(* IEC 61131-3 sources: Summary-ETFA22/benchmark/PLCopen_safety, 34 files *)

(* ---- SFAntivalent.st ---- *)
PROGRAM Main
VAR_INPUT
    Activate : BOOL;
    SChannelNC : SAFEBOOL;
    SChannelNO : SAFEBOOL;
    DiscrepancyTime : TIME;
END_VAR
VAR
    SFAntivalent : SFAntivalent;
END_VAR
SFAntivalent(Activate:=Activate,SChannelNC:=SChannelNC,SChannelNO:=SChannelNO,DiscrepancyTime:=DiscrepancyTime);
END_PROGRAM

FUNCTION_BLOCK SFAntivalent
VAR_INPUT
    Activate : BOOL;
    SChannelNC : SAFEBOOL;
    SChannelNO : SAFEBOOL;
    DiscrepancyTime : TIME;
END_VAR
VAR
    IN : BOOL;
    PT : TIME;
    running : BOOL;
    Q : BOOL;
END_VAR
VAR_OUTPUT
    Ready : BOOL;
    SAntivalentOut : BOOL;
    Error : BOOL;
    DiagCode : WORD;
END_VAR

IF NOT Activate THEN
    DiagCode := 16#0000;
ELSE
    CASE DiagCode OF
    16#0000:
        IF Activate THEN
            DiagCode := 16#8001;
        END_IF;
    16#8001:
        IF SChannelNC AND SChannelNO THEN
            DiagCode := 16#8004;
            IN:=TRUE;
            PT:=DiscrepancyTime;
            IF NOT running AND NOT Q THEN
                running := TRUE;
            ELSIF running AND NOT Q THEN
                Q := NONDETERMINISTIC_BOOL();
                running := NOT Q;
            END_IF;
        ELSIF NOT SChannelNC AND NOT SChannelNO THEN
            DiagCode := 16#8014;
            IN:=TRUE;
            PT:=DiscrepancyTime;
            IF NOT running AND NOT Q THEN
                running := TRUE;
            ELSIF running AND NOT Q THEN
                Q := NONDETERMINISTIC_BOOL();
                running := NOT Q;
            END_IF;
        ELSIF SChannelNC AND NOT SChannelNO THEN
            DiagCode := 16#8000;
        END_IF;
    16#8004:
        IF Q THEN
            DiagCode := 16#C001;
        ELSIF NOT SChannelNC THEN
            DiagCode := 16#8001;
        ELSIF NOT SChannelNO THEN
            DiagCode := 16#8000;
        END_IF;
    16#C001,
    16#C002:
        IF NOT SChannelNC AND SChannelNO THEN
            DiagCode := 16#8001;
        END_IF;
    16#8014:
        IF Q THEN
            DiagCode := 16#C002;
        ELSIF SChannelNO THEN
            DiagCode := 16#8001;
        ELSIF SChannelNC THEN
            DiagCode := 16#8000;
        END_IF;
    16#C003:
        IF NOT SChannelNC AND SChannelNO THEN
            DiagCode := 16#8001;
        END_IF;
    16#8005:
        IF Q THEN
            DiagCode := 16#C003;
        ELSIF NOT SChannelNC AND SChannelNO THEN
            DiagCode := 16#8001;
        END_IF;
    16#8000:
        IF NOT SChannelNC OR SChannelNO THEN
            DiagCode := 16#8005;
            IN:=TRUE;
            PT:=DiscrepancyTime;
            IF NOT running AND NOT Q THEN
                running := TRUE;
            ELSIF running AND NOT Q THEN
                Q := NONDETERMINISTIC_BOOL();
                running := NOT Q;
            END_IF;
        ELSIF NOT SChannelNC AND SChannelNO THEN
            DiagCode := 16#8001;
        END_IF;
    END_CASE;
END_IF;

CASE DiagCode OF
16#0000:
    Q := FALSE;
    running := FALSE;
    Ready := FALSE;
    Error := FALSE;
    SAntivalentOut:= FALSE;
16#8000:
    Q := FALSE;
    running := FALSE;
    Ready := TRUE;
    Error := FALSE;
    SAntivalentOut := TRUE;
16#8001:
    IN:=FALSE;
    PT:=DiscrepancyTime;
    Q := FALSE;
    running := FALSE;
    Ready := TRUE;
    Error := FALSE;
    SAntivalentOut:= FALSE;
16#8004,
16#8014,
16#8005:
    IN := TRUE;
    PT := DiscrepancyTime;
    IF NOT running AND NOT Q THEN
        running := TRUE;
    ELSIF running AND NOT Q THEN
        Q := NONDETERMINISTIC_BOOL();
        running := NOT Q;
    END_IF;
    Ready := TRUE;
    Error := FALSE;
    SAntivalentOut:= FALSE;
16#C001,
16#C002,
16#C003:
    IN := FALSE;
    PT := DiscrepancyTime;
    Q := FALSE;
    running := FALSE;
    Ready := TRUE;
    Error := TRUE;
    SAntivalentOut:= FALSE;
END_CASE;
END_FUNCTION_BLOCK

(* ---- SFAntivalent_CAP.st ---- *)
PROGRAM Main
VAR_INPUT
    Activate : BOOL;
    SChannelNC : SAFEBOOL;
    SChannelNO : SAFEBOOL;
    DiscrepancyTime : TIME;
END_VAR
VAR
    SFAntivalent : SFAntivalent;
END_VAR
SFAntivalent(Activate:=Activate,SChannelNC:=SChannelNC,SChannelNO:=SChannelNO,DiscrepancyTime:=DiscrepancyTime);
END_PROGRAM

FUNCTION_BLOCK SFAntivalent
VAR_INPUT
    Activate : BOOL;
    SChannelNC : SAFEBOOL;
    SChannelNO : SAFEBOOL;
    DiscrepancyTime : TIME;
END_VAR
VAR
    IN : BOOL;
    PT : TIME;
    running : BOOL;
    Q : BOOL;
END_VAR
VAR_OUTPUT
    Ready : BOOL;
    SAntivalentOut : BOOL;
    Error : BOOL;
    DiagCode : WORD;
END_VAR

IF NOT Activate THEN
    DiagCode := 16#0000;
ELSE
    CASE DiagCode OF
    change(16#0000, 16#0000):
        IF Activate THEN
            DiagCode := change(16#8001, 16#8001);
        END_IF;
    16#8001:
        IF SChannelNC AND SChannelNO THEN
            DiagCode := 16#8004;
            IN:=TRUE;
            PT:=DiscrepancyTime;
            IF NOT running AND NOT Q THEN
                running := TRUE;
            ELSIF running AND NOT Q THEN
                Q := NONDETERMINISTIC_BOOL();
                running := NOT Q;
            END_IF;
        ELSIF NOT SChannelNC AND NOT SChannelNO THEN
            DiagCode := 16#8014;
            IN:=TRUE;
            PT:=DiscrepancyTime;
            IF NOT running AND NOT Q THEN
                running := TRUE;
            ELSIF running AND NOT Q THEN
                Q := NONDETERMINISTIC_BOOL();
                running := NOT Q;
            END_IF;
        ELSIF SChannelNC AND NOT SChannelNO THEN
            DiagCode := 16#8000;
        END_IF;
    16#8004:
        IF Q THEN
            DiagCode := 16#C001;
        ELSIF NOT SChannelNC THEN
            DiagCode := 16#8001;
        ELSIF NOT SChannelNO THEN
            DiagCode := 16#8000;
        END_IF;
    16#C001,
    16#C002:
        IF NOT SChannelNC AND SChannelNO THEN
            DiagCode := 16#8001;
        END_IF;
    16#8014:
        IF Q THEN
            DiagCode := 16#C002;
        ELSIF SChannelNO THEN
            DiagCode := 16#8001;
        ELSIF SChannelNC THEN
            DiagCode := 16#8000;
        END_IF;
    16#C003:
        IF NOT SChannelNC AND SChannelNO THEN
            DiagCode := 16#8001;
        END_IF;
    16#8005:
        IF Q THEN
            DiagCode := 16#C003;
        ELSIF NOT SChannelNC AND SChannelNO THEN
            DiagCode := 16#8001;
        END_IF;
    16#8000:
        IF NOT SChannelNC OR SChannelNO THEN
            DiagCode := 16#8005;
            IN:=TRUE;
            PT:=DiscrepancyTime;
            IF NOT running AND NOT Q THEN
                running := TRUE;
            ELSIF running AND NOT Q THEN
                Q := NONDETERMINISTIC_BOOL();
                running := NOT Q;
            END_IF;
        ELSIF NOT SChannelNC AND SChannelNO THEN
            DiagCode := 16#8001;
        END_IF;
    END_CASE;
END_IF;

CASE DiagCode OF
16#0000:
    Q := FALSE;
    running := FALSE;
    Ready := FALSE;
    Error := FALSE;
    SAntivalentOut:= FALSE;
16#8000:
    Q := FALSE;
    running := FALSE;
    Ready := TRUE;
    Error := FALSE;
    SAntivalentOut := TRUE;
16#8001:
    IN:=FALSE;
    PT:=DiscrepancyTime;
    Q := FALSE;
    running := FALSE;
    Ready := TRUE;
    Error := FALSE;
    SAntivalentOut:= FALSE;
16#8004,
16#8014,
16#8005:
    IN := TRUE;
    PT := DiscrepancyTime;
    IF NOT running AND NOT Q THEN
        running := TRUE;
    ELSIF running AND NOT Q THEN
        Q := NONDETERMINISTIC_BOOL();
        running := NOT Q;
    END_IF;
    Ready := TRUE;
    Error := FALSE;
    SAntivalentOut:= FALSE;
16#C001,
16#C002,
16#C003:
    IN := FALSE;
    PT := DiscrepancyTime;
    Q := FALSE;
    running := FALSE;
    Ready := TRUE;
    Error := TRUE;
    SAntivalentOut:= FALSE;
END_CASE;
END_FUNCTION_BLOCK

(* ---- SFEDM.st ---- *)
PROGRAM Main
VAR_INPUT
    Activate : BOOL;
    SOutControl	: SAFEBOOL;
    SEDM1 : SAFEBOOL;
    SEDM2 : SAFEBOOL;
    MonitoringTime : TIME;
    SStartReset	: SAFEBOOL;
    Reset : BOOL;
END_VAR
VAR
    SFEDM : SFEDM;
END_VAR
SFEDM(Activate:=Activate,SOutControl:=SOutControl,SEDM1:=SEDM1,SEDM2:=SEDM2,MonitoringTime:=MonitoringTime,
SStartReset:=SStartReset,Reset:=Reset);
END_PROGRAM

FUNCTION_BLOCK SFEDM
VAR_INPUT
    Activate : BOOL ;
    SOutControl	: SAFEBOOL ;
    SEDM1 : SAFEBOOL ;
    SEDM2 : SAFEBOOL ;
    MonitoringTime : TIME;
    SStartReset	: SAFEBOOL ;
    Reset : BOOL ;
END_VAR
VAR
    IN : BOOL;
    PT : TIME;
    running : BOOL;
    Q : BOOL;
    RTRIGatResetQ : BOOL;
    RTRIGatResetM : BOOL;
    RTRIGatOutControlQ : BOOL;
    RTRIGatOutControlM : BOOL;
    RTRIGatEDM1Q : BOOL;
    RTRIGatEDM1M : BOOL;
    RTRIGatEDM2Q : BOOL;
    RTRIGatEDM2M : BOOL;
END_VAR
VAR_OUTPUT
    Ready : BOOL ;
    SEDMOut	: SAFEBOOL ;
    Error : BOOL ;
    DiagCode : WORD:=16#0000 ;
END_VAR
(* Rising edge detection *)
RTRIGatResetQ := Reset AND NOT RTRIGatResetM;
RTRIGatResetM := Reset;

RTRIGatOutControlQ := SOutControl AND NOT RTRIGatOutControlM;
RTRIGatOutControlM := SOutControl;

RTRIGatEDM1Q := SEDM1 AND NOT RTRIGatEDM1M;
RTRIGatEDM1M := SEDM1;

RTRIGatEDM2Q := SEDM2 AND NOT RTRIGatEDM2M;
RTRIGatEDM2M := SEDM2;

IF NOT Activate THEN
    DiagCode := 16#0000;
ELSE
    CASE DiagCode OF
    16#0000:
        IF Activate THEN
            DiagCode := 16#8001;
        END_IF;
    16#8000:
        IF Q AND SEDM1 AND NOT SEDM2 THEN
            DiagCode := 16#C070;
        ELSIF Q AND NOT SEDM1 AND SEDM2 THEN
            DiagCode := 16#C080;
        ELSIF Q AND SEDM1 AND SEDM2 THEN
            DiagCode := 16#C090;
        ELSIF NOT SOutControl THEN
            DiagCode := 16#8010;
            IN:=FALSE;
            Q := FALSE;
            running := FALSE;
        END_IF;
    16#8001:
        IF Reset AND NOT RTRIGatResetQ AND NOT SStartReset THEN
            DiagCode := 16#C001;
        ELSIF RTRIGatResetQ AND RTRIGatOutControlQ AND NOT SStartReset THEN
            DiagCode := 16#C111;
        ELSIF RTRIGatResetQ OR SStartReset THEN
            DiagCode := 16#8010;
            IN:=FALSE;
            Q := FALSE;
            running := FALSE;
        END_IF;
    16#8010:
        IF SOutControl AND NOT SEDM1 AND SEDM2 THEN
            DiagCode := 16#C010;
        ELSIF SOutControl AND SEDM1 AND NOT SEDM2 THEN
            DiagCode := 16#C020;
        ELSIF SOutControl AND NOT SEDM1 AND NOT SEDM2 THEN
            DiagCode := 16#C030;
        ELSIF Q AND NOT SEDM1 AND SEDM2 THEN
            DiagCode := 16#C040;
        ELSIF Q AND SEDM1 AND NOT SEDM2 THEN
            DiagCode := 16#C050;
        ELSIF Q AND NOT SEDM1 AND NOT SEDM2 THEN
            DiagCode := 16#C060;
        ELSIF SOutControl THEN
            DiagCode := 16#8000;
            IN:=FALSE;
            Q := FALSE;
            running := FALSE;
        END_IF;
    16#C001:
        IF NOT Reset THEN
            DiagCode := 16#8001;
        END_IF;
    16#C010, 16#C020, 16#C030:
        IF (Reset AND NOT RTRIGatResetQ AND SEDM1 AND SEDM2) OR (RTRIGatResetQ AND RTRIGatEDM1Q AND NOT RTRIGatEDM2Q) THEN
            DiagCode := 16#C011;
        ELSIF (Reset AND NOT RTRIGatResetQ AND SEDM1 AND SEDM2) OR (RTRIGatResetQ AND NOT RTRIGatEDM1Q AND RTRIGatEDM2Q) THEN
            DiagCode := 16#C021;
        ELSIF (Reset AND NOT RTRIGatResetQ AND SEDM1 AND SEDM2) OR (RTRIGatResetQ AND RTRIGatEDM1Q AND RTRIGatEDM2Q) THEN
            DiagCode := 16#C031;
        ELSIF RTRIGatResetQ AND SEDM1 AND SEDM2 THEN
            DiagCode := 16#8010;
            IN:=FALSE;
            Q := FALSE;
            running := FALSE;
        END_IF;
    16#C011:
        IF NOT Reset THEN
            DiagCode := 16#C010;
        END_IF;
    16#C021:
        IF NOT Reset THEN
            DiagCode := 16#C020;
        END_IF;
    16#C031:
        IF NOT Reset THEN
            DiagCode := 16#C030;
        END_IF;
    16#C040, 16#C050, 16#C060:
        IF (Reset AND NOT RTRIGatResetQ AND SEDM1 AND SEDM2) OR (RTRIGatResetQ AND RTRIGatEDM1Q AND NOT RTRIGatEDM2Q) THEN
            DiagCode := 16#C041;
        ELSIF (Reset AND NOT RTRIGatResetQ AND SEDM1 AND SEDM2) OR (RTRIGatResetQ AND NOT RTRIGatEDM1Q AND RTRIGatEDM2Q) THEN
            DiagCode := 16#C051;
        ELSIF (Reset AND NOT RTRIGatResetQ AND SEDM1 AND SEDM2) OR (RTRIGatResetQ AND RTRIGatEDM1Q AND RTRIGatEDM2Q) THEN
            DiagCode := 16#C061;
        ELSIF RTRIGatResetQ AND SEDM1 AND SEDM2 THEN
            DiagCode := 16#8010;
            IN:=FALSE;
            Q := FALSE;
            running := FALSE;
        END_IF;
    16#C041:
        IF NOT Reset THEN
            DiagCode := 16#C040;
        END_IF;
    16#C051:
        IF NOT Reset THEN
            DiagCode := 16#C050;
        END_IF;
    16#C061:
        IF NOT Reset THEN
            DiagCode := 16#C060;
        END_IF;
    16#C070:
        IF Reset AND NOT RTRIGatResetQ THEN
            DiagCode := 16#C071;
        ELSIF RTRIGatResetQ AND NOT (RTRIGatEDM1Q OR RTRIGatEDM2Q) THEN
            DiagCode := 16#8010;
            IN:=FALSE;
            Q := FALSE;
            running := FALSE;
        END_IF;
    16#C080:
        IF Reset AND NOT RTRIGatResetQ THEN
            DiagCode := 16#C081;
        ELSIF RTRIGatResetQ AND NOT (RTRIGatEDM1Q OR RTRIGatEDM2Q) THEN
            DiagCode := 16#8010;
            IN:=FALSE;
            Q := FALSE;
            running := FALSE;
        END_IF;
    16#C090:
        IF Reset AND NOT RTRIGatResetQ THEN
            DiagCode := 16#C091;
        ELSIF RTRIGatResetQ AND NOT (RTRIGatEDM1Q OR RTRIGatEDM2Q) THEN
            DiagCode := 16#8010;
            IN:=FALSE;
            Q := FALSE;
            running := FALSE;
        END_IF;
    16#C071:
        IF NOT Reset THEN
            DiagCode := 16#C070;
        END_IF;
    16#C081:
        IF NOT Reset THEN
            DiagCode := 16#C080;
        END_IF;
    16#C091:
        IF NOT Reset THEN
            DiagCode := 16#C090;
        END_IF;
    16#C111:
        IF NOT Reset THEN
            DiagCode := 16#8001;
        END_IF;
    END_CASE;
END_IF;
CASE DiagCode OF
16#0000:
    Ready := FALSE;
    SEDMOut := FALSE;
    Error := FALSE;
16#8001:
    Ready := TRUE;
    SEDMOut := FALSE;
    Error := FALSE;
16#8010:
    Ready := TRUE;
    SEDMOut := FALSE;
    Error := FALSE;
    IN:=TRUE;
    PT:=MonitoringTime;
    IF NOT running AND NOT Q THEN
        running := TRUE;
    ELSIF running AND NOT Q THEN
        Q := NONDETERMINISTIC_BOOL();
        running := NOT Q;
    END_IF;
16#8000:
    Ready := TRUE;
    SEDMOut := TRUE;
    Error := FALSE;
    IN:=TRUE;
    PT:=MonitoringTime;
    IF NOT running AND NOT Q THEN
        running := TRUE;
    ELSIF running AND NOT Q THEN
        Q := NONDETERMINISTIC_BOOL();
        running := NOT Q;
    END_IF;
16#C001, 16#C010, 16#C011, 16#C020, 16#C021, 16#C030, 16#C031, 16#C040, 16#C041, 16#C050, 16#C051, 16#C060, 16#C061, 16#C070, 16#C071, 16#C080, 16#C081, 16#C090, 16#C091, 16#C111:
    Ready := TRUE;
    SEDMOut := FALSE;
    Error := TRUE;
END_CASE;
END_FUNCTION_BLOCK

FUNCTION_BLOCK RTRIG
VAR_INPUT
    CLK : BOOL;
END_VAR
VAR
    M : BOOL;
END_VAR
VAR_OUTPUT
    Q : BOOL;
END_VAR
    Q := CLK AND NOT M;
    M := CLK;
END_FUNCTION_BLOCK

(* ---- SFEDM_CAP.st ---- *)
PROGRAM Main
VAR_INPUT
    Activate : BOOL;
    SOutControl	: SAFEBOOL;
    SEDM1 : SAFEBOOL;
    SEDM2 : SAFEBOOL;
    MonitoringTime : TIME;
    SStartReset	: SAFEBOOL;
    Reset : BOOL;
END_VAR
VAR
    SFEDM : SFEDM;
END_VAR
SFEDM(Activate:=Activate,SOutControl:=SOutControl,SEDM1:=SEDM1,SEDM2:=SEDM2,MonitoringTime:=MonitoringTime,
SStartReset:=SStartReset,Reset:=Reset);
END_PROGRAM

FUNCTION_BLOCK SFEDM
VAR_INPUT
    Activate : BOOL ;
    SOutControl	: SAFEBOOL ;
    SEDM1 : SAFEBOOL ;
    SEDM2 : SAFEBOOL ;
    MonitoringTime : TIME;
    SStartReset	: SAFEBOOL ;
    Reset : BOOL ;
END_VAR
VAR
    IN : BOOL;
    PT : TIME;
    running : BOOL;
    Q : BOOL;
    RTRIGatResetQ : BOOL;
    RTRIGatResetM : BOOL;
    RTRIGatOutControlQ : BOOL;
    RTRIGatOutControlM : BOOL;
    RTRIGatEDM1Q : BOOL;
    RTRIGatEDM1M : BOOL;
    RTRIGatEDM2Q : BOOL;
    RTRIGatEDM2M : BOOL;
END_VAR
VAR_OUTPUT
    Ready : BOOL ;
    SEDMOut	: SAFEBOOL ;
    Error : BOOL ;
    DiagCode : WORD:=16#0000 ;
END_VAR
(* Rising edge detection *)
RTRIGatResetQ := Reset AND NOT RTRIGatResetM;
RTRIGatResetM := Reset;

RTRIGatOutControlQ := SOutControl AND NOT RTRIGatOutControlM;
RTRIGatOutControlM := SOutControl;

RTRIGatEDM1Q := SEDM1 AND NOT RTRIGatEDM1M;
RTRIGatEDM1M := SEDM1;

RTRIGatEDM2Q := SEDM2 AND NOT RTRIGatEDM2M;
RTRIGatEDM2M := SEDM2;

IF NOT Activate THEN
    DiagCode := change(16#0000, 16#8001);
ELSE
    CASE DiagCode OF
    16#0000:
        IF Activate THEN
            DiagCode := 16#8001;
        END_IF;
    16#8000:
        IF Q AND SEDM1 AND NOT SEDM2 THEN
            DiagCode := 16#C070;
        ELSIF Q AND NOT SEDM1 AND SEDM2 THEN
            DiagCode := 16#C080;
        ELSIF Q AND SEDM1 AND SEDM2 THEN
            DiagCode := 16#C090;
        ELSIF NOT SOutControl THEN
            DiagCode := 16#8010;
            IN:=FALSE;
            Q := FALSE;
            running := FALSE;
        END_IF;
    16#8001:
        IF Reset AND NOT RTRIGatResetQ AND NOT SStartReset THEN
            DiagCode := 16#C001;
        ELSIF RTRIGatResetQ AND RTRIGatOutControlQ AND NOT SStartReset THEN
            DiagCode := 16#C111;
        ELSIF RTRIGatResetQ OR SStartReset THEN
            DiagCode := 16#8010;
            IN:=FALSE;
            Q := FALSE;
            running := FALSE;
        END_IF;
    16#8010:
        IF SOutControl AND NOT SEDM1 AND SEDM2 THEN
            DiagCode := 16#C010;
        ELSIF SOutControl AND SEDM1 AND NOT SEDM2 THEN
            DiagCode := 16#C020;
        ELSIF SOutControl AND NOT SEDM1 AND NOT SEDM2 THEN
            DiagCode := 16#C030;
        ELSIF Q AND NOT SEDM1 AND SEDM2 THEN
            DiagCode := 16#C040;
        ELSIF Q AND SEDM1 AND NOT SEDM2 THEN
            DiagCode := 16#C050;
        ELSIF Q AND NOT SEDM1 AND NOT SEDM2 THEN
            DiagCode := 16#C060;
        ELSIF SOutControl THEN
            DiagCode := 16#8000;
            IN:=FALSE;
            Q := FALSE;
            running := FALSE;
        END_IF;
    16#C001:
        IF NOT Reset THEN
            DiagCode := 16#8001;
        END_IF;
    16#C010, 16#C020, 16#C030:
        IF (Reset AND NOT RTRIGatResetQ AND SEDM1 AND SEDM2) OR (RTRIGatResetQ AND RTRIGatEDM1Q AND NOT RTRIGatEDM2Q) THEN
            DiagCode := 16#C011;
        ELSIF (Reset AND NOT RTRIGatResetQ AND SEDM1 AND SEDM2) OR (RTRIGatResetQ AND NOT RTRIGatEDM1Q AND RTRIGatEDM2Q) THEN
            DiagCode := 16#C021;
        ELSIF (Reset AND NOT RTRIGatResetQ AND SEDM1 AND SEDM2) OR (RTRIGatResetQ AND RTRIGatEDM1Q AND RTRIGatEDM2Q) THEN
            DiagCode := 16#C031;
        ELSIF RTRIGatResetQ AND SEDM1 AND SEDM2 THEN
            DiagCode := 16#8010;
            IN:=FALSE;
            Q := FALSE;
            running := FALSE;
        END_IF;
    16#C011:
        IF NOT Reset THEN
            DiagCode := 16#C010;
        END_IF;
    16#C021:
        IF NOT Reset THEN
            DiagCode := 16#C020;
        END_IF;
    16#C031:
        IF NOT Reset THEN
            DiagCode := 16#C030;
        END_IF;
    16#C040, 16#C050, 16#C060:
        IF (Reset AND NOT RTRIGatResetQ AND SEDM1 AND SEDM2) OR (RTRIGatResetQ AND RTRIGatEDM1Q AND NOT RTRIGatEDM2Q) THEN
            DiagCode := 16#C041;
        ELSIF (Reset AND NOT RTRIGatResetQ AND SEDM1 AND SEDM2) OR (RTRIGatResetQ AND NOT RTRIGatEDM1Q AND RTRIGatEDM2Q) THEN
            DiagCode := 16#C051;
        ELSIF (Reset AND NOT RTRIGatResetQ AND SEDM1 AND SEDM2) OR (RTRIGatResetQ AND RTRIGatEDM1Q AND RTRIGatEDM2Q) THEN
            DiagCode := 16#C061;
        ELSIF RTRIGatResetQ AND SEDM1 AND SEDM2 THEN
            DiagCode := 16#8010;
            IN:=FALSE;
            Q := FALSE;
            running := FALSE;
        END_IF;
    16#C041:
        IF NOT Reset THEN
            DiagCode := 16#C040;
        END_IF;
    16#C051:
        IF NOT Reset THEN
            DiagCode := 16#C050;
        END_IF;
    16#C061:
        IF NOT Reset THEN
            DiagCode := 16#C060;
        END_IF;
    16#C070:
        IF Reset AND NOT RTRIGatResetQ THEN
            DiagCode := 16#C071;
        ELSIF RTRIGatResetQ AND NOT (RTRIGatEDM1Q OR RTRIGatEDM2Q) THEN
            DiagCode := 16#8010;
            IN:=FALSE;
            Q := FALSE;
            running := FALSE;
        END_IF;
    16#C080:
        IF Reset AND NOT RTRIGatResetQ THEN
            DiagCode := 16#C081;
        ELSIF RTRIGatResetQ AND NOT (RTRIGatEDM1Q OR RTRIGatEDM2Q) THEN
            DiagCode := 16#8010;
            IN:=FALSE;
            Q := FALSE;
            running := FALSE;
        END_IF;
    16#C090:
        IF Reset AND NOT RTRIGatResetQ THEN
            DiagCode := 16#C091;
        ELSIF RTRIGatResetQ AND NOT (RTRIGatEDM1Q OR RTRIGatEDM2Q) THEN
            DiagCode := 16#8010;
            IN:=FALSE;
            Q := FALSE;
            running := FALSE;
        END_IF;
    16#C071:
        IF NOT Reset THEN
            DiagCode := 16#C070;
        END_IF;
    16#C081:
        IF NOT Reset THEN
            DiagCode := 16#C080;
        END_IF;
    16#C091:
        IF NOT Reset THEN
            DiagCode := 16#C090;
        END_IF;
    16#C111:
        IF NOT Reset THEN
            DiagCode := 16#8001;
        END_IF;
    END_CASE;
END_IF;
CASE DiagCode OF
16#0000:
    Ready := FALSE;
    SEDMOut := FALSE;
    Error := FALSE;
16#8001:
    Ready := TRUE;
    SEDMOut := FALSE;
    Error := FALSE;
16#8010:
    Ready := TRUE;
    SEDMOut := FALSE;
    Error := FALSE;
    IN:=TRUE;
    PT:=MonitoringTime;
    IF NOT running AND NOT Q THEN
        running := TRUE;
    ELSIF running AND NOT Q THEN
        Q := NONDETERMINISTIC_BOOL();
        running := NOT Q;
    END_IF;
16#8000:
    Ready := TRUE;
    SEDMOut := TRUE;
    Error := FALSE;
    IN:=TRUE;
    PT:=MonitoringTime;
    IF NOT running AND NOT Q THEN
        running := TRUE;
    ELSIF running AND NOT Q THEN
        Q := NONDETERMINISTIC_BOOL();
        running := NOT Q;
    END_IF;
16#C001, 16#C010, 16#C011, 16#C020, 16#C021, 16#C030, 16#C031, 16#C040, 16#C041, 16#C050, 16#C051, 16#C060, 16#C061, 16#C070, 16#C071, 16#C080, 16#C081, 16#C090, 16#C091, 16#C111:
    Ready := TRUE;
    SEDMOut := FALSE;
    Error := TRUE;
END_CASE;
END_FUNCTION_BLOCK

FUNCTION_BLOCK RTRIG
VAR_INPUT
    CLK : BOOL;
END_VAR
VAR
    M : BOOL;
END_VAR
VAR_OUTPUT
    Q : BOOL;
END_VAR
    Q := CLK AND NOT M;
    M := CLK;
END_FUNCTION_BLOCK

(* ---- SFEmergencyStop.st ---- *)
PROGRAM Main
VAR_INPUT
    Activate : BOOL;
    SEStopIn : BOOL;
    SStartReset : BOOL;
    SAutoReset : BOOL;
    Reset : BOOL;
END_VAR
VAR
    SFEmergencyStop : SFEmergencyStop;
END_VAR
SFEmergencyStop(Activate:=Activate,SEStopIn:=SEStopIn,SStartReset:=SStartReset,SAutoReset:=SAutoReset,Reset:=Reset);
END_PROGRAM

FUNCTION_BLOCK SFEmergencyStop
VAR_INPUT
    Activate : BOOL;
    SEStopIn : BOOL;
    SStartReset : BOOL;
    SAutoReset : BOOL;
    Reset : BOOL;
END_VAR
VAR
    RTRIGatResetQ : BOOL;
    RTRIGatResetM : BOOL;
END_VAR
VAR_OUTPUT
    Ready : BOOL;
    SEStopOut : BOOL;
    Error : BOOL;
    DiagCode : WORD;
END_VAR
RTRIGatResetQ := Reset AND NOT RTRIGatResetM;
RTRIGatResetM := Reset;

IF NOT Activate THEN
    DiagCode := 16#0000;
ELSE
    CASE DiagCode OF
    16#0000:
        IF Activate THEN
            DiagCode := 16#8001;
        END_IF;
    16#8001:
        IF NOT SStartReset THEN
            DiagCode := 16#8002;
        ELSIF SStartReset AND NOT SEStopIn THEN
            DiagCode := 16#8004;
        ELSIF SEStopIn AND SStartReset THEN
            DiagCode := 16#8000;
        END_IF;
    16#8002:
        IF SEStopIn THEN
            DiagCode := 16#8003;
        END_IF;
    16#8003:
        IF Reset AND NOT RTRIGatResetQ THEN
            DiagCode := 16#C001;
        ELSIF NOT SEStopIn THEN
            DiagCode := 16#8002;
        ELSIF RTRIGatResetQ THEN
            DiagCode := 16#8000;
        END_IF;
    16#C001:
        IF NOT Reset THEN
            DiagCode := 16#8003;
        END_IF;
    16#8004:
        IF SEStopIn AND NOT SAutoReset THEN
            DiagCode := 16#8005;
        ELSIF SEStopIn AND SAutoReset THEN
            DiagCode := 16#8000;
        END_IF;
    16#8005:
        IF Reset AND NOT RTRIGatResetQ THEN
            DiagCode := 16#C002;
        ELSIF NOT SEStopIn THEN
            DiagCode := 16#8004;
        ELSIF RTRIGatResetQ OR SAutoReset THEN
            DiagCode := 16#8000;
        END_IF;
    16#C002:
        IF NOT Reset THEN
            DiagCode := 16#8005;
        END_IF;
    16#8000:
        IF NOT SEStopIn THEN
            DiagCode := 16#8004;
        END_IF;
    END_CASE;
END_IF;
CASE DiagCode OF
16#0000:
    Ready := FALSE;
    Error := FALSE;
    SEStopOut := FALSE;
16#8001:
    Ready := TRUE;
    Error := FALSE;
    SEStopOut := FALSE;
16#8002:
    Ready := TRUE;
    Error := FALSE;
    SEStopOut := FALSE;
16#8003:
    Ready := TRUE;
    Error := FALSE;
    SEStopOut := FALSE;
16#C001:
    Ready := TRUE;
    Error := TRUE;
    SEStopOut := FALSE;
16#8004:
    Ready := TRUE;
    Error := FALSE;
    SEStopOut := FALSE;
16#8005:
    Ready := TRUE;
    Error := FALSE;
    SEStopOut := FALSE;
16#C002:
    Ready := TRUE;
    Error := TRUE;
    SEStopOut := FALSE;
16#8000:
    Ready := TRUE;
    Error := FALSE;
    SEStopOut := TRUE;
END_CASE;
END_FUNCTION_BLOCK

(* ---- SFEmergencyStop_CAP.st ---- *)
PROGRAM Main
VAR_INPUT
    Activate : BOOL;
    SEStopIn : BOOL;
    SStartReset : BOOL;
    SAutoReset : BOOL;
    Reset : BOOL;
END_VAR
VAR
    SFEmergencyStop : SFEmergencyStop;
END_VAR
SFEmergencyStop(Activate:=Activate,SEStopIn:=SEStopIn,SStartReset:=SStartReset,SAutoReset:=SAutoReset,Reset:=Reset);
END_PROGRAM

FUNCTION_BLOCK SFEmergencyStop
VAR_INPUT
    Activate : BOOL;
    SEStopIn : BOOL;
    SStartReset : BOOL;
    SAutoReset : BOOL;
    Reset : BOOL;
END_VAR
VAR
    RTRIGatResetQ : BOOL;
    RTRIGatResetM : BOOL;
END_VAR
VAR_OUTPUT
    Ready : BOOL;
    SEStopOut : BOOL;
    Error : BOOL;
    DiagCode : WORD;
END_VAR
RTRIGatResetQ := Reset AND NOT RTRIGatResetM;
RTRIGatResetM := Reset;

IF NOT Activate THEN
    DiagCode := change(16#0000, 16#8001);
ELSE
    CASE DiagCode OF
    16#0000:
        IF Activate THEN
            DiagCode := 16#8001;
        END_IF;
    16#8001:
        IF NOT SStartReset THEN
            DiagCode := 16#8002;
        ELSIF SStartReset AND NOT SEStopIn THEN
            DiagCode := 16#8004;
        ELSIF SEStopIn AND SStartReset THEN
            DiagCode := 16#8000;
        END_IF;
    16#8002:
        IF SEStopIn THEN
            DiagCode := 16#8003;
        END_IF;
    16#8003:
        IF Reset AND NOT RTRIGatResetQ THEN
            DiagCode := 16#C001;
        ELSIF NOT SEStopIn THEN
            DiagCode := 16#8002;
        ELSIF RTRIGatResetQ THEN
            DiagCode := 16#8000;
        END_IF;
    16#C001:
        IF NOT Reset THEN
            DiagCode := 16#8003;
        END_IF;
    16#8004:
        IF SEStopIn AND NOT SAutoReset THEN
            DiagCode := 16#8005;
        ELSIF SEStopIn AND SAutoReset THEN
            DiagCode := 16#8000;
        END_IF;
    16#8005:
        IF Reset AND NOT RTRIGatResetQ THEN
            DiagCode := 16#C002;
        ELSIF NOT SEStopIn THEN
            DiagCode := 16#8004;
        ELSIF RTRIGatResetQ OR SAutoReset THEN
            DiagCode := 16#8000;
        END_IF;
    16#C002:
        IF NOT Reset THEN
            DiagCode := 16#8005;
        END_IF;
    16#8000:
        IF NOT SEStopIn THEN
            DiagCode := 16#8004;
        END_IF;
    END_CASE;
END_IF;
CASE DiagCode OF
16#0000:
    Ready := FALSE;
    Error := FALSE;
    SEStopOut := FALSE;
16#8001:
    Ready := TRUE;
    Error := FALSE;
    SEStopOut := FALSE;
16#8002:
    Ready := TRUE;
    Error := FALSE;
    SEStopOut := FALSE;
16#8003:
    Ready := TRUE;
    Error := FALSE;
    SEStopOut := FALSE;
16#C001:
    Ready := TRUE;
    Error := TRUE;
    SEStopOut := FALSE;
16#8004:
    Ready := TRUE;
    Error := FALSE;
    SEStopOut := FALSE;
16#8005:
    Ready := TRUE;
    Error := FALSE;
    SEStopOut := FALSE;
16#C002:
    Ready := TRUE;
    Error := TRUE;
    SEStopOut := FALSE;
16#8000:
    Ready := TRUE;
    Error := FALSE;
    SEStopOut := TRUE;
END_CASE;
END_FUNCTION_BLOCK

(* ---- SFEnableSwitch.st ---- *)
PROGRAM Main
VAR_INPUT
    Activate : BOOL;
    SSafetyActive : SAFEBOOL;
    SEnableSwitchCh1 : SAFEBOOL;
    SEnableSwitchCh2 : SAFEBOOL;
    SAutoReset : SAFEBOOL;
    Reset : BOOL;
END_VAR
VAR
    SFEnableSwitch : SFEnableSwitch;
END_VAR
SFEnableSwitch(Activate:=Activate,SSafetyActive:=SSafetyActive,SEnableSwitchCh1:=SEnableSwitchCh1,
SEnableSwitchCh2:=SEnableSwitchCh2,SAutoReset:=SAutoReset,Reset:=Reset);
END_PROGRAM

FUNCTION_BLOCK SFEnableSwitch
VAR_INPUT
    Activate : BOOL;
    SSafetyActive : SAFEBOOL;
    SEnableSwitchCh1 : SAFEBOOL;
    SEnableSwitchCh2 : SAFEBOOL;
    SAutoReset : SAFEBOOL;
    Reset : BOOL;
END_VAR
VAR
    RTRIGatResetQ : BOOL;
    RTRIGatResetM : BOOL;
END_VAR
VAR_OUTPUT
    Ready : BOOL;
    SEnableSwitchOut : SAFEBOOL;
    Error : BOOL;
    DiagCode : WORD;
END_VAR
RTRIGatResetQ := Reset AND NOT RTRIGatResetM;
RTRIGatResetM := Reset;

IF NOT Activate THEN
    DiagCode := 16#0000;
ELSIF NOT SSafetyActive THEN
    DiagCode := 16#8004;
ELSE
    CASE DiagCode OF
    16#0000:
        IF Activate THEN
            DiagCode := 16#8004;
        END_IF;
    16#8000:
        IF (NOT (SEnableSwitchCh1 OR SEnableSwitchCh2)) OR (SEnableSwitchCh1 AND NOT SEnableSwitchCh2) THEN
            DiagCode := 16#8007;
        ELSIF NOT SEnableSwitchCh1 AND SEnableSwitchCh2 THEN
            DiagCode := 16#8006;
        END_IF;
    16#8004:
        IF SSafetyActive THEN
            DiagCode := 16#8005;
        END_IF;
    16#8005:
        IF NOT (NOT SEnableSwitchCh1 AND SEnableSwitchCh2) THEN
            DiagCode := 16#C010;
        ELSIF NOT SEnableSwitchCh1 AND SEnableSwitchCh2 THEN
            DiagCode := 16#8006;
        END_IF;
    16#8006:
        IF SEnableSwitchCh1 AND SEnableSwitchCh2 THEN
            DiagCode := 16#8000;
        ELSIF (NOT (SEnableSwitchCh1 OR SEnableSwitchCh2)) OR (SEnableSwitchCh1 AND NOT SEnableSwitchCh2) THEN
            DiagCode := 16#8007;
        END_IF;
    16#8007:
        IF SEnableSwitchCh1 AND SEnableSwitchCh2 THEN
            DiagCode := 16#C030;
        ELSIF NOT SEnableSwitchCh1 AND SEnableSwitchCh2 THEN
            DiagCode := 16#8006;
        END_IF;
    16#C001:
        IF NOT Reset THEN
            DiagCode := 16#C020;
        END_IF;
    16#C002:
        IF NOT Reset THEN
            DiagCode := 16#C040;
        END_IF;
    16#C010:
        IF NOT SEnableSwitchCh1 AND SEnableSwitchCh2 THEN
            DiagCode := 16#C020;
        END_IF;
    16#C020:
        IF NOT (NOT SEnableSwitchCh1 AND SEnableSwitchCh2) THEN
            DiagCode := 16#C010;
        ELSIF Reset AND NOT RTRIGatResetQ AND NOT SAutoReset THEN
            DiagCode := 16#C001;
        ELSIF RTRIGatResetQ OR SAutoReset THEN
            DiagCode := 16#8006;
        END_IF;
    16#C030:
        IF NOT (SEnableSwitchCh1 AND SEnableSwitchCh2) THEN
            DiagCode := 16#C040;
        END_IF;
    16#C040:
        IF SEnableSwitchCh1 AND SEnableSwitchCh2 THEN
            DiagCode := 16#C030;
        ELSIF Reset AND RTRIGatResetQ AND NOT SAutoReset THEN
            DiagCode := 16#C002;
        ELSIF RTRIGatResetQ OR SAutoReset THEN
            DiagCode := 16#8007;
        END_IF;
    END_CASE;
END_IF;

CASE DiagCode OF
16#C001,
16#C002,
16#C010,
16#C020,
16#C030,
16#C040:
    Ready := TRUE;
    SEnableSwitchOut := FALSE;
    Error := TRUE;
16#0000:
    Ready := FALSE;
    SEnableSwitchOut := FALSE;
    Error := FALSE;
16#8000:
    Ready := TRUE;
    SEnableSwitchOut := TRUE;
    Error := FALSE;
16#8004,
16#8005,
16#8006,
16#8007:
    Ready := TRUE;
    SEnableSwitchOut := FALSE;
    Error := FALSE;
END_CASE;
END_FUNCTION_BLOCK

(* ---- SFEnableSwitch_CAP.st ---- *)
PROGRAM Main
VAR_INPUT
    Activate : BOOL;
    SSafetyActive : SAFEBOOL;
    SEnableSwitchCh1 : SAFEBOOL;
    SEnableSwitchCh2 : SAFEBOOL;
    SAutoReset : SAFEBOOL;
    Reset : BOOL;
END_VAR
VAR
    SFEnableSwitch : SFEnableSwitch;
END_VAR
SFEnableSwitch(Activate:=Activate,SSafetyActive:=SSafetyActive,SEnableSwitchCh1:=SEnableSwitchCh1,
SEnableSwitchCh2:=SEnableSwitchCh2,SAutoReset:=SAutoReset,Reset:=Reset);
END_PROGRAM

FUNCTION_BLOCK SFEnableSwitch
VAR_INPUT
    Activate : BOOL;
    SSafetyActive : SAFEBOOL;
    SEnableSwitchCh1 : SAFEBOOL;
    SEnableSwitchCh2 : SAFEBOOL;
    SAutoReset : SAFEBOOL;
    Reset : BOOL;
END_VAR
VAR
    RTRIGatResetQ : BOOL;
    RTRIGatResetM : BOOL;
END_VAR
VAR_OUTPUT
    Ready : BOOL;
    SEnableSwitchOut : SAFEBOOL;
    Error : BOOL;
    DiagCode : WORD;
END_VAR
RTRIGatResetQ := Reset AND NOT RTRIGatResetM;
RTRIGatResetM := Reset;

IF NOT Activate THEN
    DiagCode := 16#0000;
ELSIF NOT SSafetyActive THEN
    DiagCode := 16#8004;
ELSE
    CASE DiagCode OF
    16#0000:
        IF Activate THEN
            DiagCode := change(16#8004, 16#8004);
        END_IF;
    16#8000:
        IF (NOT (SEnableSwitchCh1 OR SEnableSwitchCh2)) OR (SEnableSwitchCh1 AND NOT SEnableSwitchCh2) THEN
            DiagCode := 16#8007;
        ELSIF NOT SEnableSwitchCh1 AND SEnableSwitchCh2 THEN
            DiagCode := 16#8006;
        END_IF;
    16#8004:
        IF SSafetyActive THEN
            DiagCode := 16#8005;
        END_IF;
    16#8005:
        IF NOT (NOT SEnableSwitchCh1 AND SEnableSwitchCh2) THEN
            DiagCode := 16#C010;
        ELSIF NOT SEnableSwitchCh1 AND SEnableSwitchCh2 THEN
            DiagCode := 16#8006;
        END_IF;
    16#8006:
        IF SEnableSwitchCh1 AND SEnableSwitchCh2 THEN
            DiagCode := 16#8000;
        ELSIF (NOT (SEnableSwitchCh1 OR SEnableSwitchCh2)) OR (SEnableSwitchCh1 AND NOT SEnableSwitchCh2) THEN
            DiagCode := 16#8007;
        END_IF;
    16#8007:
        IF SEnableSwitchCh1 AND SEnableSwitchCh2 THEN
            DiagCode := 16#C030;
        ELSIF NOT SEnableSwitchCh1 AND SEnableSwitchCh2 THEN
            DiagCode := 16#8006;
        END_IF;
    16#C001:
        IF NOT Reset THEN
            DiagCode := 16#C020;
        END_IF;
    16#C002:
        IF NOT Reset THEN
            DiagCode := 16#C040;
        END_IF;
    16#C010:
        IF NOT SEnableSwitchCh1 AND SEnableSwitchCh2 THEN
            DiagCode := 16#C020;
        END_IF;
    16#C020:
        IF NOT (NOT SEnableSwitchCh1 AND SEnableSwitchCh2) THEN
            DiagCode := 16#C010;
        ELSIF Reset AND NOT RTRIGatResetQ AND NOT SAutoReset THEN
            DiagCode := 16#C001;
        ELSIF RTRIGatResetQ OR SAutoReset THEN
            DiagCode := 16#8006;
        END_IF;
    16#C030:
        IF NOT (SEnableSwitchCh1 AND SEnableSwitchCh2) THEN
            DiagCode := 16#C040;
        END_IF;
    16#C040:
        IF SEnableSwitchCh1 AND SEnableSwitchCh2 THEN
            DiagCode := 16#C030;
        ELSIF Reset AND RTRIGatResetQ AND NOT SAutoReset THEN
            DiagCode := 16#C002;
        ELSIF RTRIGatResetQ OR SAutoReset THEN
            DiagCode := 16#8007;
        END_IF;
    END_CASE;
END_IF;

CASE DiagCode OF
16#C001,
16#C002,
16#C010,
16#C020,
16#C030,
16#C040:
    Ready := TRUE;
    SEnableSwitchOut := FALSE;
    Error := TRUE;
16#0000:
    Ready := FALSE;
    SEnableSwitchOut := FALSE;
    Error := FALSE;
16#8000:
    Ready := TRUE;
    SEnableSwitchOut := TRUE;
    Error := FALSE;
16#8004,
16#8005,
16#8006,
16#8007:
    Ready := TRUE;
    SEnableSwitchOut := FALSE;
    Error := FALSE;
END_CASE;
END_FUNCTION_BLOCK

(* ---- SFEquivalent.st ---- *)
PROGRAM Main
VAR_INPUT
    Activate : BOOL;
    SChannelA : BOOL;
    SChannelB : BOOL;
    DiscrepancyTime : TIME;
END_VAR
VAR
    SFEquivalent : SFEquivalent;
END_VAR
SFEquivalent(Activate:=Activate,SChannelA:=SChannelA,SChannelB:=SChannelB,DiscrepancyTime:=DiscrepancyTime);
END_PROGRAM

FUNCTION_BLOCK SFEquivalent
VAR_INPUT
    Activate : BOOL;
    SChannelA : BOOL;
    SChannelB : BOOL;
    DiscrepancyTime : TIME;
END_VAR
VAR
    IN : BOOL;
    PT : TIME;
    running : BOOL;
    Q : BOOL;
END_VAR
VAR_OUTPUT
    Ready : BOOL;
	SEquivalentOut : BOOL;
	Error : BOOL;
	DiagCode : WORD;
END_VAR

IF NOT Activate THEN
    DiagCode := 16#0000;
ELSE
    CASE DiagCode OF
    16#0000:
        IF Activate THEN
            DiagCode := 16#8001;
        END_IF;
    16#8001:
        IF SChannelA AND NOT SChannelB THEN
            DiagCode := 16#8004;
        ELSIF SChannelB AND NOT SChannelA THEN
            DiagCode := 16#8014;
        ELSIF SChannelA AND SChannelB THEN
            DiagCode := 16#8000;
        END_IF;
    16#8004:
        IF Q THEN
            DiagCode := 16#C001;
        ELSIF NOT SChannelA THEN
            DiagCode := 16#8001;
        ELSIF SChannelB THEN
            DiagCode := 16#8000;
        END_IF;
    16#C001,
    16#C002:
        IF NOT SChannelA AND NOT SChannelB THEN
            DiagCode := 16#8001;
        END_IF;
    16#8014:
        IF Q THEN
            DiagCode := 16#C002;
        ELSIF NOT SChannelB THEN
            DiagCode := 16#8001;
        ELSIF SChannelA THEN
            DiagCode := 16#8000;
        END_IF;
    16#C003:
        IF NOT SChannelA AND NOT SChannelB THEN
            DiagCode := 16#8001;
        END_IF;
    16#8005:
        IF Q THEN
            DiagCode := 16#C003;
        ELSIF NOT SChannelA AND NOT SChannelB THEN
            DiagCode := 16#8001;
        END_IF;
    16#8000:
        IF SChannelA XOR SChannelB THEN
            DiagCode := 16#8005;
        ELSIF NOT SChannelA AND NOT SChannelB THEN
            DiagCode := 16#8001;
        END_IF;
    END_CASE;
END_IF;

CASE DiagCode OF
16#0000:
    IN:=FALSE;
    PT:=DiscrepancyTime;
    Q := FALSE;
    running := FALSE;
    Ready := FALSE;
    Error := FALSE;
    SEquivalentOut:= FALSE;
16#8000:
    IN:=FALSE;
    PT:=DiscrepancyTime;
    Q := FALSE;
    running := FALSE;
    Ready := TRUE;
    Error := FALSE;
    SEquivalentOut := TRUE;
16#8001:
    IN:=FALSE;
    PT:=DiscrepancyTime;
    Q := FALSE;
    running := FALSE;
    Ready := TRUE;
    Error := FALSE;
    SEquivalentOut:= FALSE;
16#8004,
16#8014,
16#8005:
	IN:=TRUE;
	PT:=DiscrepancyTime;
	IF NOT running AND NOT Q THEN
        running := TRUE;
    ELSIF running AND NOT Q THEN
        Q := NONDETERMINISTIC_BOOL();
        running := NOT Q;
    END_IF;
    Ready := TRUE;
    Error := FALSE;
    SEquivalentOut:= FALSE;
16#C001,
16#C002,
16#C003:
    IN:=FALSE;
    PT:=DiscrepancyTime;
    Q := FALSE;
    running := FALSE;
    Ready := TRUE;
    Error := TRUE;
    SEquivalentOut:= FALSE;
END_CASE;
END_FUNCTION_BLOCK

(* ---- SFEquivalent_CAP.st ---- *)
PROGRAM Main
VAR_INPUT
    Activate : BOOL;
    SChannelA : BOOL;
    SChannelB : BOOL;
    DiscrepancyTime : TIME;
END_VAR
VAR
    SFEquivalent : SFEquivalent;
END_VAR
SFEquivalent(Activate:=Activate,SChannelA:=SChannelA,SChannelB:=SChannelB,DiscrepancyTime:=DiscrepancyTime);
END_PROGRAM

FUNCTION_BLOCK SFEquivalent
VAR_INPUT
    Activate : BOOL;
    SChannelA : BOOL;
    SChannelB : BOOL;
    DiscrepancyTime : TIME;
END_VAR
VAR
    IN : BOOL;
    PT : TIME;
    running : BOOL;
    Q : BOOL;
END_VAR
VAR_OUTPUT
    Ready : BOOL;
	SEquivalentOut : BOOL;
	Error : BOOL;
	DiagCode : WORD;
END_VAR

IF NOT Activate THEN
    DiagCode := 16#0000;
ELSE
    CASE DiagCode OF
    16#0000:
        IF Activate THEN
            DiagCode := 16#8001;
        END_IF;
    16#8001:
        IF SChannelA AND NOT SChannelB THEN
            DiagCode := 16#8004;
        ELSIF SChannelB AND NOT SChannelA THEN
            DiagCode := 16#8014;
        ELSIF SChannelA AND SChannelB THEN
            DiagCode := 16#8000;
        END_IF;
    16#8004:
        IF Q THEN
            DiagCode := 16#C001;
        ELSIF NOT SChannelA THEN
            DiagCode := 16#8001;
        ELSIF SChannelB THEN
            DiagCode := change(16#8000, 16#8004);
        END_IF;
    16#C001,
    16#C002:
        IF NOT SChannelA AND NOT SChannelB THEN
            DiagCode := 16#8001;
        END_IF;
    16#8014:
        IF Q THEN
            DiagCode := 16#C002;
        ELSIF NOT SChannelB THEN
            DiagCode := 16#8001;
        ELSIF SChannelA THEN
            DiagCode := 16#8000;
        END_IF;
    16#C003:
        IF NOT SChannelA AND NOT SChannelB THEN
            DiagCode := 16#8001;
        END_IF;
    16#8005:
        IF Q THEN
            DiagCode := 16#C003;
        ELSIF NOT SChannelA AND NOT SChannelB THEN
            DiagCode := 16#8001;
        END_IF;
    16#8000:
        IF SChannelA XOR SChannelB THEN
            DiagCode := 16#8005;
        ELSIF NOT SChannelA AND NOT SChannelB THEN
            DiagCode := 16#8001;
        END_IF;
    END_CASE;
END_IF;

CASE DiagCode OF
16#0000:
    IN:=FALSE;
    PT:=DiscrepancyTime;
    Q := FALSE;
    running := FALSE;
    Ready := FALSE;
    Error := FALSE;
    SEquivalentOut:= FALSE;
16#8000:
    IN:=FALSE;
    PT:=DiscrepancyTime;
    Q := FALSE;
    running := FALSE;
    Ready := TRUE;
    Error := FALSE;
    SEquivalentOut := TRUE;
16#8001:
    IN:=FALSE;
    PT:=DiscrepancyTime;
    Q := FALSE;
    running := FALSE;
    Ready := TRUE;
    Error := FALSE;
    SEquivalentOut:= FALSE;
16#8004,
16#8014,
16#8005:
	IN:=TRUE;
	PT:=DiscrepancyTime;
	IF NOT running AND NOT Q THEN
        running := TRUE;
    ELSIF running AND NOT Q THEN
        Q := NONDETERMINISTIC_BOOL();
        running := NOT Q;
    END_IF;
    Ready := TRUE;
    Error := FALSE;
    SEquivalentOut:= FALSE;
16#C001,
16#C002,
16#C003:
    IN:=FALSE;
    PT:=DiscrepancyTime;
    Q := FALSE;
    running := FALSE;
    Ready := TRUE;
    Error := TRUE;
    SEquivalentOut:= FALSE;
END_CASE;
END_FUNCTION_BLOCK

(* ---- SFESPE.st ---- *)
PROGRAM Main
VAR_INPUT
    Activate : BOOL;
    SESPEIn : BOOL;
    SStartReset : BOOL;
    SAutoReset : BOOL;
    Reset : BOOL;
END_VAR
VAR
    SFESPE : SFESPE;
END_VAR
SFESPE(Activate:=Activate,SESPEIn:=SESPEIn,SStartReset:=SStartReset,SAutoReset:=SAutoReset,Reset:=Reset);
END_PROGRAM

FUNCTION_BLOCK SFESPE
VAR_INPUT
    Activate : BOOL;
    SESPEIn : BOOL;
    SStartReset : BOOL;
    SAutoReset : BOOL;
    Reset : BOOL;
END_VAR
VAR
    RTRIGatResetQ : BOOL;
    RTRIGatResetM : BOOL;
END_VAR
VAR_OUTPUT
    Ready : BOOL;
    SESPEOut : BOOL;
    Error : BOOL;
    DiagCode : WORD;
END_VAR
RTRIGatResetQ := Reset AND NOT RTRIGatResetM;
RTRIGatResetM := Reset;
IF NOT Activate THEN
    DiagCode := 16#0000;
ELSE
    CASE DiagCode OF
    16#0000:
        IF Activate THEN
            DiagCode := 16#8001;
        END_IF;
    16#8001:
        IF NOT SStartReset THEN
            DiagCode := 16#8002;
        ELSIF SStartReset AND NOT SESPEIn THEN
            DiagCode := 16#8004;
        ELSIF SESPEIn AND SStartReset THEN
            DiagCode := 16#8000;
        END_IF;
    16#8002:
        IF SESPEIn THEN
            DiagCode := 16#8003;
        END_IF;
    16#8003:
        IF Reset AND NOT RTRIGatResetQ THEN
            DiagCode := 16#C001;
        ELSIF NOT SESPEIn THEN
            DiagCode := 16#8002;
        ELSIF RTRIGatResetQ THEN
            DiagCode := 16#8000;
        END_IF;
    16#C001:
        IF NOT Reset THEN
            DiagCode := 16#8003;
        END_IF;
    16#8004:
        IF SESPEIn AND NOT SAutoReset THEN
            DiagCode := 16#8005;
        ELSIF SESPEIn AND SAutoReset THEN
            DiagCode := 16#8000;
        END_IF;
    16#8005:
        IF Reset AND NOT RTRIGatResetQ THEN
            DiagCode := 16#C002;
        ELSIF NOT SESPEIn THEN
            DiagCode := 16#8004;
        ELSIF RTRIGatResetQ OR SAutoReset THEN
            DiagCode := 16#8000;
        END_IF;
    16#C002:
        IF NOT Reset THEN
            DiagCode := 16#8005;
        END_IF;
    16#8000:
        IF NOT SESPEIn THEN
            DiagCode := 16#8004;
        END_IF;
    END_CASE;
END_IF;
CASE DiagCode OF
16#0000:
    Ready := FALSE;
    Error := FALSE;
    SESPEOut := FALSE;
16#8001:
    Ready := TRUE;
    Error := FALSE;
    SESPEOut := FALSE;
16#8002:
    Ready := TRUE;
    Error := FALSE;
    SESPEOut := FALSE;
16#8003:
    Ready := TRUE;
    Error := FALSE;
    SESPEOut := FALSE;
16#C001:
    Ready := TRUE;
    Error := TRUE;
    SESPEOut := FALSE;
16#8004:
    Ready := TRUE;
    Error := FALSE;
    SESPEOut := FALSE;
16#8005:
    Ready := TRUE;
    Error := FALSE;
    SESPEOut := FALSE;
16#C002:
    Ready := TRUE;
    Error := TRUE;
    SESPEOut := FALSE;
16#8000:
    Ready := TRUE;
    Error := FALSE;
    SESPEOut := TRUE;
END_CASE;
END_FUNCTION_BLOCK

(* ---- SFESPE_CAP.st ---- *)
PROGRAM Main
VAR_INPUT
    Activate : BOOL;
    SESPEIn : BOOL;
    SStartReset : BOOL;
    SAutoReset : BOOL;
    Reset : BOOL;
END_VAR
VAR
    SFESPE : SFESPE;
END_VAR
SFESPE(Activate:=Activate,SESPEIn:=SESPEIn,SStartReset:=SStartReset,SAutoReset:=SAutoReset,Reset:=Reset);
END_PROGRAM

FUNCTION_BLOCK SFESPE
VAR_INPUT
    Activate : BOOL;
    SESPEIn : BOOL;
    SStartReset : BOOL;
    SAutoReset : BOOL;
    Reset : BOOL;
END_VAR
VAR
    RTRIGatResetQ : BOOL;
    RTRIGatResetM : BOOL;
END_VAR
VAR_OUTPUT
    Ready : BOOL;
    SESPEOut : BOOL;
    Error : BOOL;
    DiagCode : WORD;
END_VAR
RTRIGatResetQ := Reset AND NOT RTRIGatResetM;
RTRIGatResetM := Reset;
IF NOT Activate THEN
    DiagCode := 16#0000;
ELSE
    CASE DiagCode OF
    16#0000:
        IF Activate THEN
            DiagCode := change(16#8001, 16#8004);
        END_IF;
    16#8001:
        IF NOT SStartReset THEN
            DiagCode := 16#8002;
        ELSIF SStartReset AND NOT SESPEIn THEN
            DiagCode := 16#8004;
        ELSIF SESPEIn AND SStartReset THEN
            DiagCode := 16#8000;
        END_IF;
    16#8002:
        IF SESPEIn THEN
            DiagCode := 16#8003;
        END_IF;
    16#8003:
        IF Reset AND NOT RTRIGatResetQ THEN
            DiagCode := 16#C001;
        ELSIF NOT SESPEIn THEN
            DiagCode := 16#8002;
        ELSIF RTRIGatResetQ THEN
            DiagCode := 16#8000;
        END_IF;
    16#C001:
        IF NOT Reset THEN
            DiagCode := 16#8003;
        END_IF;
    16#8004:
        IF SESPEIn AND NOT SAutoReset THEN
            DiagCode := 16#8005;
        ELSIF SESPEIn AND SAutoReset THEN
            DiagCode := 16#8000;
        END_IF;
    16#8005:
        IF Reset AND NOT RTRIGatResetQ THEN
            DiagCode := 16#C002;
        ELSIF NOT SESPEIn THEN
            DiagCode := 16#8004;
        ELSIF RTRIGatResetQ OR SAutoReset THEN
            DiagCode := 16#8000;
        END_IF;
    16#C002:
        IF NOT Reset THEN
            DiagCode := 16#8005;
        END_IF;
    16#8000:
        IF NOT SESPEIn THEN
            DiagCode := change(16#8004, 16#8000);
        END_IF;
    END_CASE;
END_IF;
CASE DiagCode OF
16#0000:
    Ready := FALSE;
    Error := FALSE;
    SESPEOut := FALSE;
16#8001:
    Ready := TRUE;
    Error := FALSE;
    SESPEOut := FALSE;
16#8002:
    Ready := TRUE;
    Error := FALSE;
    SESPEOut := FALSE;
16#8003:
    Ready := TRUE;
    Error := FALSE;
    SESPEOut := FALSE;
16#C001:
    Ready := TRUE;
    Error := TRUE;
    SESPEOut := FALSE;
16#8004:
    Ready := TRUE;
    Error := FALSE;
    SESPEOut := FALSE;
16#8005:
    Ready := TRUE;
    Error := FALSE;
    SESPEOut := FALSE;
16#C002:
    Ready := TRUE;
    Error := TRUE;
    SESPEOut := FALSE;
16#8000:
    Ready := TRUE;
    Error := FALSE;
    SESPEOut := TRUE;
END_CASE;
END_FUNCTION_BLOCK

(* ---- SFGuardLocking.st ---- *)
PROGRAM Main
VAR_INPUT
    Activate : BOOL;
    SGuardMonitoring : SAFEBOOL;
    SSafetyActive : SAFEBOOL;
    SGuardLock : SAFEBOOL;
    UnlockRequest : BOOL;
    SStartReset : SAFEBOOL;
    SAutoReset : SAFEBOOL;
    Reset : BOOL;
END_VAR
VAR
    SFGuardLocking : SFGuardLocking;
END_VAR
SFGuardLocking(Activate:=Activate,SGuardMonitoring:=SGuardMonitoring,SSafetyActive:=SSafetyActive,SGuardLock:=SGuardLock,
UnlockRequest:=UnlockRequest,SStartReset:=SStartReset,SAutoReset:=SAutoReset,Reset:=Reset);
END_PROGRAM

FUNCTION_BLOCK SFGuardLocking
VAR_INPUT
    Activate : BOOL;
    SGuardMonitoring : SAFEBOOL;
    SSafetyActive : SAFEBOOL;
    SGuardLock : SAFEBOOL;
    UnlockRequest : BOOL;
    SStartReset : SAFEBOOL;
    SAutoReset : SAFEBOOL;
    Reset : BOOL;
END_VAR
VAR
    RTRIGatResetQ : BOOL;
    RTRIGatResetM : BOOL;
    RTRIGatUnlockRequestQ : BOOL;
    RTRIGatUnlockRequestM : BOOL;
END_VAR
VAR_OUTPUT
    Ready : BOOL;
    SGuardLocked : SAFEBOOL;
    SUnlockGuard : SAFEBOOL;
    Error : BOOL;
    DiagCode : WORD;
END_VAR
RTRIGatResetQ := Reset AND NOT RTRIGatResetM;
RTRIGatResetM := Reset;

RTRIGatUnlockRequestQ := UnlockRequest AND NOT RTRIGatUnlockRequestM;
RTRIGatUnlockRequestM := UnlockRequest;

IF NOT Activate THEN
    DiagCode := 16#0000;
END_IF;
CASE DiagCode OF
16#0000:
    IF Activate THEN
        DiagCode := 16#8001;
    END_IF;
16#8000:
    IF NOT SGuardLock OR NOT SGuardMonitoring THEN
        DiagCode := 16#C004;
    ELSIF RTRIGatUnlockRequestQ AND SSafetyActive THEN
        DiagCode := 16#8013;
    END_IF;
16#8001:
    IF Reset AND NOT RTRIGatResetQ AND NOT SStartReset THEN
        DiagCode := 16#C001;
    ELSIF NOT SGuardLock OR NOT SGuardMonitoring THEN
        DiagCode := 16#8011;
    ELSIF (RTRIGatResetQ OR SStartReset) AND SGuardMonitoring AND SGuardLock THEN
        DiagCode := 16#8000;
    END_IF;
16#8003:
    IF Reset AND NOT RTRIGatResetQ AND NOT SAutoReset THEN
        DiagCode := 16#C003;
    ELSIF NOT SGuardMonitoring OR NOT SGuardLock THEN
        DiagCode := 16#8011;
    ELSIF RTRIGatResetQ OR SAutoReset THEN
        DiagCode := 16#8000;
    END_IF;
16#8011:
    IF NOT SSafetyActive AND (NOT SGuardMonitoring OR NOT SGuardLock) THEN
        DiagCode := 16#C004;
    ELSIF (SSafetyActive AND UnlockRequest) OR NOT SGuardMonitoring THEN
        DiagCode := 16#8012;
    ELSIF SGuardMonitoring AND SGuardLock THEN
        DiagCode := 16#8003;
    END_IF;
16#8012:
    IF SGuardMonitoring THEN
        DiagCode := 16#8013;
    ELSIF NOT SSafetyActive AND NOT SGuardMonitoring THEN
        DiagCode := 16#C004;
    END_IF;
16#8013:
    IF NOT SGuardMonitoring THEN
        DiagCode := 16#8012;
    ELSIF NOT UnlockRequest THEN
        DiagCode := 16#8011;
    END_IF;
16#8014:
    IF Reset AND NOT RTRIGatResetQ THEN
        DiagCode := 16#C002;
    ELSIF NOT SSafetyActive THEN
        DiagCode := 16#C004;
    ELSIF RTRIGatResetQ THEN
        DiagCode := 16#8011;
    END_IF;
16#C001:
    IF NOT Reset THEN
        DiagCode := 16#8001;
    END_IF;
16#C002:
    IF NOT Reset THEN
        DiagCode := 16#8014;
    END_IF;
16#C003:
    IF NOT Reset THEN
        DiagCode := 16#8003;
    END_IF;
16#C004:
    IF SSafetyActive THEN
        DiagCode := 16#8014;
    END_IF;
END_CASE;
CASE DiagCode OF
16#0000:
    Ready := FALSE;
    SGuardLocked := FALSE;
    SUnlockGuard := FALSE;
    Error := FALSE;
16#8000:
    Ready := TRUE;
    SGuardLocked := TRUE;
    SUnlockGuard := FALSE;
    Error := FALSE;
16#8001,
16#8003,
16#8011,
16#8014:
    Ready := TRUE;
    SGuardLocked := FALSE;
    SUnlockGuard := FALSE;
    Error := FALSE;
16#8012,
16#8013:
    Ready := TRUE;
    SGuardLocked := FALSE;
    SUnlockGuard := TRUE;
    Error := FALSE;
16#C001,
16#C002,
16#C003,
16#C004:
    Ready := TRUE;
    SGuardLocked := FALSE;
    SUnlockGuard := FALSE;
    Error := TRUE;
END_CASE;
END_FUNCTION_BLOCK

(* ---- SFGuardLocking_CAP.st ---- *)
PROGRAM Main
VAR_INPUT
    Activate : BOOL;
    SGuardMonitoring : SAFEBOOL;
    SSafetyActive : SAFEBOOL;
    SGuardLock : SAFEBOOL;
    UnlockRequest : BOOL;
    SStartReset : SAFEBOOL;
    SAutoReset : SAFEBOOL;
    Reset : BOOL;
END_VAR
VAR
    SFGuardLocking : SFGuardLocking;
END_VAR
SFGuardLocking(Activate:=Activate,SGuardMonitoring:=SGuardMonitoring,SSafetyActive:=SSafetyActive,SGuardLock:=SGuardLock,
UnlockRequest:=UnlockRequest,SStartReset:=SStartReset,SAutoReset:=SAutoReset,Reset:=Reset);
END_PROGRAM

FUNCTION_BLOCK SFGuardLocking
VAR_INPUT
    Activate : BOOL;
    SGuardMonitoring : SAFEBOOL;
    SSafetyActive : SAFEBOOL;
    SGuardLock : SAFEBOOL;
    UnlockRequest : BOOL;
    SStartReset : SAFEBOOL;
    SAutoReset : SAFEBOOL;
    Reset : BOOL;
END_VAR
VAR
    RTRIGatResetQ : BOOL;
    RTRIGatResetM : BOOL;
    RTRIGatUnlockRequestQ : BOOL;
    RTRIGatUnlockRequestM : BOOL;
END_VAR
VAR_OUTPUT
    Ready : BOOL;
    SGuardLocked : SAFEBOOL;
    SUnlockGuard : SAFEBOOL;
    Error : BOOL;
    DiagCode : WORD;
END_VAR
RTRIGatResetQ := Reset AND NOT RTRIGatResetM;
RTRIGatResetM := Reset;

RTRIGatUnlockRequestQ := UnlockRequest AND NOT RTRIGatUnlockRequestM;
RTRIGatUnlockRequestM := UnlockRequest;

IF NOT Activate THEN
    DiagCode := 16#0000;
END_IF;
CASE DiagCode OF
16#0000:
    IF Activate THEN
        DiagCode := 16#8001;
    END_IF;
16#8000:
    IF NOT SGuardLock OR NOT SGuardMonitoring THEN
        DiagCode := 16#C004;
    ELSIF RTRIGatUnlockRequestQ AND SSafetyActive THEN
        DiagCode := 16#8013;
    END_IF;
16#8001:
    IF Reset AND NOT RTRIGatResetQ AND NOT SStartReset THEN
        DiagCode := 16#C001;
    ELSIF NOT SGuardLock OR NOT SGuardMonitoring THEN
        DiagCode := 16#8011;
    ELSIF (RTRIGatResetQ OR SStartReset) AND SGuardMonitoring AND SGuardLock THEN
        DiagCode := 16#8000;
    END_IF;
16#8003:
    IF change(Reset AND NOT RTRIGatResetQ AND NOT SAutoReset, TRUE) THEN
        DiagCode := 16#C003;
    ELSIF NOT SGuardMonitoring OR NOT SGuardLock THEN
        DiagCode := 16#8011;
    ELSIF RTRIGatResetQ OR SAutoReset THEN
        DiagCode := 16#8000;
    END_IF;
16#8011:
    IF NOT SSafetyActive AND (NOT SGuardMonitoring OR NOT SGuardLock) THEN
        DiagCode := 16#C004;
    ELSIF (SSafetyActive AND UnlockRequest) OR NOT SGuardMonitoring THEN
        DiagCode := 16#8012;
    ELSIF SGuardMonitoring AND SGuardLock THEN
        DiagCode := 16#8003;
    END_IF;
16#8012:
    IF SGuardMonitoring THEN
        DiagCode := 16#8013;
    ELSIF NOT SSafetyActive AND NOT SGuardMonitoring THEN
        DiagCode := 16#C004;
    END_IF;
16#8013:
    IF NOT SGuardMonitoring THEN
        DiagCode := 16#8012;
    ELSIF NOT UnlockRequest THEN
        DiagCode := 16#8011;
    END_IF;
16#8014:
    IF Reset AND NOT RTRIGatResetQ THEN
        DiagCode := 16#C002;
    ELSIF NOT SSafetyActive THEN
        DiagCode := 16#C004;
    ELSIF RTRIGatResetQ THEN
        DiagCode := 16#8011;
    END_IF;
16#C001:
    IF NOT Reset THEN
        DiagCode := 16#8001;
    END_IF;
16#C002:
    IF NOT Reset THEN
        DiagCode := 16#8014;
    END_IF;
16#C003:
    IF NOT Reset THEN
        DiagCode := 16#8003;
    END_IF;
16#C004:
    IF SSafetyActive THEN
        DiagCode := 16#8014;
    END_IF;
END_CASE;
CASE DiagCode OF
16#0000:
    Ready := FALSE;
    SGuardLocked := FALSE;
    SUnlockGuard := FALSE;
    Error := FALSE;
16#8000:
    Ready := TRUE;
    SGuardLocked := TRUE;
    SUnlockGuard := FALSE;
    Error := FALSE;
16#8001,
16#8003,
16#8011,
16#8014:
    Ready := TRUE;
    SGuardLocked := FALSE;
    SUnlockGuard := FALSE;
    Error := FALSE;
16#8012,
16#8013:
    Ready := TRUE;
    SGuardLocked := FALSE;
    SUnlockGuard := TRUE;
    Error := FALSE;
16#C001,
16#C002,
16#C003,
16#C004:
    Ready := TRUE;
    SGuardLocked := FALSE;
    SUnlockGuard := FALSE;
    Error := TRUE;
END_CASE;
END_FUNCTION_BLOCK

(* ---- SFGuardMonitoring.st ---- *)
PROGRAM Main
VAR_INPUT
    Activate : BOOL := FALSE;
    SGuardSwitch1 : SAFEBOOL := FALSE;
    SGuardSwitch2 : SAFEBOOL := FALSE;
    DiscrepancyTime : TIME := T#0s;
    SStartReset : SAFEBOOL := FALSE;
    SAutoReset : SAFEBOOL := FALSE;
    Reset : BOOL := FALSE;
END_VAR
VAR
    SFGuardMonitoring : SFGuardMonitoring;
END_VAR
SFGuardMonitoring(Activate:=Activate,SGuardSwitch1:=SGuardSwitch1,SGuardSwitch2:=SGuardSwitch2,DiscrepancyTime:=DiscrepancyTime,
                  SStartReset:=SStartReset,SAutoReset:=SAutoReset,Reset:=Reset);
END_PROGRAM

FUNCTION_BLOCK SFGuardMonitoring
VAR_INPUT
    Activate : BOOL := FALSE;
    SGuardSwitch1 : SAFEBOOL := FALSE;
    SGuardSwitch2 : SAFEBOOL := FALSE;
    DiscrepancyTime : TIME := T#0s;
    SStartReset : SAFEBOOL := FALSE;
    SAutoReset : SAFEBOOL := FALSE;
    Reset : BOOL := FALSE;
END_VAR
VAR
    IN : BOOL;
    PT : TIME;
    running : BOOL;
    Q : BOOL;
    RTRIGatResetQ : BOOL;
    RTRIGatResetM : BOOL;
END_VAR
VAR_OUTPUT
    Ready : BOOL := FALSE;
    SGuardMonitoring : BOOL := FALSE;
    Error : BOOL := FALSE;
    DiagCode : WORD := 16#0000;
END_VAR
RTRIGatResetQ := Reset AND NOT RTRIGatResetM;
RTRIGatResetM := Reset;

IF NOT Activate THEN
    DiagCode := 16#0000;
ELSE
    CASE DiagCode OF
    16#0000:
        IF Activate THEN
            DiagCode := 16#8001;
        END_IF;
    16#8001:
        IF NOT SGuardSwitch1 OR NOT SGuardSwitch2 THEN
            DiagCode := 16#8002;
        ELSIF SGuardSwitch1 AND SGuardSwitch2 AND NOT SStartReset THEN
            DiagCode := 16#8003;
        ELSIF SGuardSwitch1 AND SGuardSwitch2 AND SStartReset THEN
            DiagCode := 16#8000;
        END_IF;
    16#8002:
        IF NOT SGuardSwitch1 AND NOT SGuardSwitch2 THEN
            DiagCode := 16#8012;
        END_IF;
    16#8003:
        IF Reset AND NOT RTRIGatResetQ THEN
            DiagCode := 16#C001;
        ELSIF NOT SGuardSwitch1 OR NOT SGuardSwitch2 THEN
            DiagCode := 16#8002;
        ELSIF RTRIGatResetQ THEN
            DiagCode := 16#8000;
        END_IF;
    16#8012:
        IF SGuardSwitch1 THEN
            DiagCode := 16#8004;
        ELSIF SGuardSwitch2 THEN
            DiagCode := 16#8014;
        END_IF;
    16#8004:
        IF Q THEN
            DiagCode := 16#C011;
        ELSIF NOT SGuardSwitch1 THEN
            DiagCode := 16#8002;
        ELSIF SGuardSwitch2 THEN
            DiagCode := 16#8005;
        END_IF;
    16#8014:
        IF Q THEN
            DiagCode := 16#C012;
        ELSIF NOT SGuardSwitch2 THEN
            DiagCode := 16#8002;
        ELSIF SGuardSwitch1 THEN
            DiagCode := 16#8005;
        END_IF;
    16#8005:
        IF NOT SGuardSwitch1 OR NOT SGuardSwitch2 THEN
            DiagCode := 16#8002;
        ELSIF NOT SAutoReset THEN
            DiagCode := 16#8003;
        ELSIF SAutoReset THEN
            DiagCode := 16#8000;
        END_IF;
    16#8000:
        IF NOT SGuardSwitch1 OR NOT SGuardSwitch2 THEN
            DiagCode := 16#8002;
        END_IF;
    16#C001:
        IF NOT Reset THEN
            DiagCode := 16#8003;
        END_IF;
    16#C011:
        IF NOT SGuardSwitch1 AND NOT SGuardSwitch2 THEN
            DiagCode := 16#8012;
        END_IF;
    16#C012:
        IF NOT SGuardSwitch1 AND NOT SGuardSwitch2 THEN
            DiagCode := 16#8012;
        END_IF;
    END_CASE;
END_IF;
CASE DiagCode OF
16#0000:
    IN:=FALSE;
    PT:=DiscrepancyTime;
    Q := FALSE;
    running := FALSE;
    Ready := FALSE;
    Error := FALSE;
    SGuardMonitoring := FALSE;
16#8000:
    IN:=FALSE;
    PT:=DiscrepancyTime;
    Q := FALSE;
    running := FALSE;
    Ready := TRUE;
    Error := FALSE;
    SGuardMonitoring  := TRUE;
16#8001,
16#8002,
16#8003,
16#8012,
16#8005:
    IN:=FALSE;
    PT:=DiscrepancyTime;
    Q := FALSE;
    running := FALSE;
    Ready := TRUE;
    Error := FALSE;
    SGuardMonitoring := FALSE;
16#8004,
16#8014:
    IN:=TRUE;
    PT:=DiscrepancyTime;
    IF NOT running AND NOT Q THEN
        running := TRUE;
    ELSIF running AND NOT Q THEN
        Q := NONDETERMINISTIC_BOOL();
        running := NOT Q;
    END_IF;
    Ready := TRUE;
    Error := FALSE;
    SGuardMonitoring := FALSE;
16#C001,
16#C011,
16#C012:
    IN:=FALSE;
    PT:=DiscrepancyTime;
    Q := FALSE;
    running := FALSE;
    Ready := TRUE;
    Error := TRUE;
    SGuardMonitoring := FALSE;
END_CASE;
END_FUNCTION_BLOCK

(* ---- SFGuardMonitoring_CAP.st ---- *)
PROGRAM Main
VAR_INPUT
    Activate : BOOL := FALSE;
    SGuardSwitch1 : SAFEBOOL := FALSE;
    SGuardSwitch2 : SAFEBOOL := FALSE;
    DiscrepancyTime : TIME := T#0s;
    SStartReset : SAFEBOOL := FALSE;
    SAutoReset : SAFEBOOL := FALSE;
    Reset : BOOL := FALSE;
END_VAR
VAR
    SFGuardMonitoring : SFGuardMonitoring;
END_VAR
SFGuardMonitoring(Activate:=Activate,SGuardSwitch1:=SGuardSwitch1,SGuardSwitch2:=SGuardSwitch2,DiscrepancyTime:=DiscrepancyTime,
                  SStartReset:=SStartReset,SAutoReset:=SAutoReset,Reset:=Reset);
END_PROGRAM

FUNCTION_BLOCK SFGuardMonitoring
VAR_INPUT
    Activate : BOOL := FALSE;
    SGuardSwitch1 : SAFEBOOL := FALSE;
    SGuardSwitch2 : SAFEBOOL := FALSE;
    DiscrepancyTime : TIME := T#0s;
    SStartReset : SAFEBOOL := FALSE;
    SAutoReset : SAFEBOOL := FALSE;
    Reset : BOOL := FALSE;
END_VAR
VAR
    IN : BOOL;
    PT : TIME;
    running : BOOL;
    Q : BOOL;
    RTRIGatResetQ : BOOL;
    RTRIGatResetM : BOOL;
END_VAR
VAR_OUTPUT
    Ready : BOOL := FALSE;
    SGuardMonitoring : BOOL := FALSE;
    Error : BOOL := FALSE;
    DiagCode : WORD := 16#0000;
END_VAR
RTRIGatResetQ := Reset AND NOT RTRIGatResetM;
RTRIGatResetM := Reset;

IF NOT Activate THEN
    DiagCode := 16#0000;
ELSE
    CASE DiagCode OF
    16#0000:
        IF Activate THEN
            DiagCode := 16#8001;
        END_IF;
    16#8001:
        IF NOT SGuardSwitch1 OR NOT SGuardSwitch2 THEN
            DiagCode := 16#8002;
        ELSIF SGuardSwitch1 AND SGuardSwitch2 AND NOT SStartReset THEN
            DiagCode := 16#8003;
        ELSIF SGuardSwitch1 AND SGuardSwitch2 AND SStartReset THEN
            DiagCode := 16#8000;
        END_IF;
    16#8002:
        IF NOT SGuardSwitch1 AND NOT SGuardSwitch2 THEN
            DiagCode := 16#8012;
        END_IF;
    16#8003:
        IF Reset AND NOT RTRIGatResetQ THEN
            DiagCode := 16#C001;
        ELSIF NOT SGuardSwitch1 OR NOT SGuardSwitch2 THEN
            DiagCode := 16#8002;
        ELSIF RTRIGatResetQ THEN
            DiagCode := 16#8000;
        END_IF;
    16#8012:
        IF SGuardSwitch1 THEN
            DiagCode := 16#8004;
        ELSIF SGuardSwitch2 THEN
            DiagCode := 16#8014;
        END_IF;
    16#8004:
        IF Q THEN
            DiagCode := 16#C011;
        ELSIF NOT SGuardSwitch1 THEN
            DiagCode := 16#8002;
        ELSIF SGuardSwitch2 THEN
            DiagCode := 16#8005;
        END_IF;
    16#8014:
        IF change(Q, FALSE) THEN
            DiagCode := 16#C012;
        ELSIF NOT SGuardSwitch2 THEN
            DiagCode := 16#8002;
        ELSIF SGuardSwitch1 THEN
            DiagCode := 16#8005;
        END_IF;
    16#8005:
        IF NOT SGuardSwitch1 OR NOT SGuardSwitch2 THEN
            DiagCode := 16#8002;
        ELSIF NOT SAutoReset THEN
            DiagCode := 16#8003;
        ELSIF SAutoReset THEN
            DiagCode := change(16#8000, 16#8001);
        END_IF;
    16#8000:
        IF NOT SGuardSwitch1 OR NOT SGuardSwitch2 THEN
            DiagCode := 16#8002;
        END_IF;
    16#C001:
        IF NOT Reset THEN
            DiagCode := 16#8003;
        END_IF;
    16#C011:
        IF NOT SGuardSwitch1 AND NOT SGuardSwitch2 THEN
            DiagCode := 16#8012;
        END_IF;
    16#C012:
        IF NOT SGuardSwitch1 AND NOT SGuardSwitch2 THEN
            DiagCode := 16#8012;
        END_IF;
    END_CASE;
END_IF;
CASE DiagCode OF
16#0000:
    IN:=FALSE;
    PT:=DiscrepancyTime;
    Q := FALSE;
    running := FALSE;
    Ready := FALSE;
    Error := FALSE;
    SGuardMonitoring := FALSE;
16#8000:
    IN:=FALSE;
    PT:=DiscrepancyTime;
    Q := FALSE;
    running := FALSE;
    Ready := TRUE;
    Error := FALSE;
    SGuardMonitoring  := TRUE;
16#8001,
16#8002,
16#8003,
16#8012,
16#8005:
    IN:=FALSE;
    PT:=DiscrepancyTime;
    Q := FALSE;
    running := FALSE;
    Ready := TRUE;
    Error := FALSE;
    SGuardMonitoring := FALSE;
16#8004,
16#8014:
    IN:=TRUE;
    PT:=DiscrepancyTime;
    IF NOT running AND NOT Q THEN
        running := TRUE;
    ELSIF running AND NOT Q THEN
        Q := NONDETERMINISTIC_BOOL();
        running := NOT Q;
    END_IF;
    Ready := TRUE;
    Error := FALSE;
    SGuardMonitoring := FALSE;
16#C001,
16#C011,
16#C012:
    IN:=FALSE;
    PT:=DiscrepancyTime;
    Q := FALSE;
    running := FALSE;
    Ready := TRUE;
    Error := TRUE;
    SGuardMonitoring := FALSE;
END_CASE;
END_FUNCTION_BLOCK

(* ---- SFModeSelector.st ---- *)
PROGRAM Main
VAR_INPUT
    Activate : BOOL;
    SMode0 : BOOL;
    SMode1 : BOOL;
    SMode2 : BOOL;
    SMode3 : BOOL;
    SMode4 : BOOL;
    SMode5 : BOOL;
    SMode6 : BOOL;
    SMode7 : BOOL;
    SUnlock : BOOL;
    SSetMode : BOOL;
    AutoSetMode : BOOL;
    ModeMonitorTime : TIME;
    Reset : BOOL;
END_VAR
VAR
    SFModeSelector : SFModeSelector;
END_VAR
SFModeSelector(Activate:=Activate,SMode0:=SMode0,SMode1:=SMode1,SMode2:=SMode2,SMode3:=SMode3,SMode4:=SMode4,SMode5:=SMode5,
SMode6:=SMode6,SMode7:=SMode7,SUnlock:=SUnlock,SSetMode:=SSetMode,AutoSetMode:=AutoSetMode,ModeMonitorTime:=ModeMonitorTime,
Reset:=Reset);
END_PROGRAM

FUNCTION_BLOCK SFModeSelector
VAR_INPUT
    Activate : BOOL;
    SMode0 : BOOL;
    SMode1 : BOOL;
    SMode2 : BOOL;
    SMode3 : BOOL;
    SMode4 : BOOL;
    SMode5 : BOOL;
    SMode6 : BOOL;
    SMode7 : BOOL;
    SUnlock : BOOL;
    SSetMode : BOOL;
    AutoSetMode : BOOL;
    ModeMonitorTime : TIME;
    Reset : BOOL;
END_VAR
VAR
    IN : BOOL;
    PT : TIME;
    running : BOOL;
    Q : BOOL;
    RTRIGatResetQ : BOOL;
    RTRIGatResetM : BOOL;
    RTRIGatSetModeQ : BOOL;
    RTRIGatSetModeM : BOOL;
    FTRIGatModeSel0Q : BOOL;
    FTRIGatModeSel0M : BOOL;
    RTRIGatModeSel0Q: BOOL;
    RTRIGatModeSel0M: BOOL;
    fallingEdgeDetected : BOOL;
END_VAR
VAR_TEMP
    Error1 : BOOL;
    Error2 : BOOL;
END_VAR
VAR_OUTPUT
    Ready : BOOL;
    SMode0Sel : BOOL;
    SMode1Sel : BOOL;
    SMode2Sel : BOOL;
    SMode3Sel : BOOL;
    SMode4Sel : BOOL;
    SMode5Sel : BOOL;
    SMode6Sel : BOOL;
    SMode7Sel : BOOL;
    SAnyModeSel : BOOL;
    Error : BOOL;
    DiagCode : WORD;
END_VAR
RTRIGatResetQ := Reset AND NOT RTRIGatResetM;
RTRIGatResetM := Reset;

RTRIGatSetModeQ := SSetMode AND NOT RTRIGatSetModeM;
RTRIGatSetModeM := SSetMode;

IF NOT Activate THEN
    DiagCode := 16#0000;
ELSE
    IF (SMode0 + SMode1 + SMode2 + SMode3 + SMode4 + SMode5 + SMode6 + SMode7 > 1) THEN
        Error1 := true;
    ELSE
        Error1 := false;
    END_IF;
    CASE DiagCode OF
    16#0000:
        IF Activate THEN
            DiagCode := 16#8005;
        END_IF;
    16#8005:
        IF (NOT SMode0 AND NOT SMode1 AND NOT SMode2 AND NOT SMode3 AND NOT SMode4 AND NOT SMode5 AND NOT SMode6 AND NOT SMode7) THEN
            FTRIGatModeSel0Q := NOT false AND FTRIGatModeSel0M;
            FTRIGatModeSel0M := false;
            RTRIGatModeSel0Q := false AND NOT RTRIGatModeSel0M;
            RTRIGatModeSel0M := false;
        ELSE
            FTRIGatModeSel0Q := NOT true AND FTRIGatModeSel0M;
            FTRIGatModeSel0M := true;
            RTRIGatModeSel0Q := true AND NOT RTRIGatModeSel0M;
            RTRIGatModeSel0M := true;
        END_IF;
        IF FTRIGatModeSel0Q THEN
            fallingEdgeDetected := TRUE;
        END_IF;
        IF fallingEdgeDetected THEN
            IN:=TRUE;
            PT:=ModeMonitorTime;
            IF NOT running AND NOT Q THEN
                running := TRUE;
            ELSIF running AND NOT Q THEN
                Q := NONDETERMINISTIC_BOOL();
                running := NOT Q;
            END_IF;
        ELSIF RTRIGatModeSel0Q THEN
            IN:=FALSE;
            PT:=ModeMonitorTime;
            Q := FALSE;
            running := FALSE;
            fallingEdgeDetected := FALSE;
        END_IF;
        Error2 := Q;
        IF Error1 THEN
            DiagCode := 16#C001;
        ELSIF Error2 THEN
            DiagCode := 16#C002;
        ELSIF ((AutoSetMode OR RTRIGatSetModeQ) AND SUnlock AND (SMode0 + SMode1 + SMode2 + SMode3 + SMode4 + SMode5 + SMode6 + SMode7 = 1)) THEN
            DiagCode := 16#8000;
        END_IF;
    16#8000:
        IF Error1 THEN
            DiagCode := 16#C001;
        ELSIF (SMode0 <> SMode0Sel OR SMode1 <> SMode1Sel OR SMode2 <> SMode2Sel OR SMode3 <> SMode3Sel
              OR SMode4 <> SMode4Sel OR SMode5 <> SMode5Sel OR SMode6 <> SMode6Sel OR SMode7 <> SMode7Sel) THEN
            DiagCode := 16#8005;
            fallingEdgeDetected := FALSE;
        ELSIF (NOT SUnlock) THEN
            DiagCode := 16#8004;
        END_IF;
    16#8004:
        IF SUnlock THEN
            DiagCode := 16#8000;
        END_IF;
    16#C001:
        IF Reset AND NOT RTRIGatResetQ THEN
            DiagCode := 16#C003;
        ELSIF RTRIGatResetQ THEN
            DiagCode := 16#8005;
            fallingEdgeDetected := FALSE;
        END_IF;
    16#C002:
        IF Reset AND NOT RTRIGatResetQ THEN
            DiagCode := 16#C004;
        ELSIF RTRIGatResetQ THEN
            DiagCode := 16#8005;
            fallingEdgeDetected := FALSE;
        END_IF;
    16#C003:
        IF (NOT Reset) THEN
            DiagCode := 16#C001;
        END_IF;
    16#C004:
        IF (NOT Reset) THEN
            DiagCode := 16#C002;
        END_IF;
    END_CASE;
END_IF;

CASE DiagCode OF
16#0000:
    Ready := false;
    SMode0Sel := false;
    SMode1Sel := false;
    SMode2Sel := false;
    SMode3Sel := false;
    SMode4Sel := false;
    SMode5Sel := false;
    SMode6Sel := false;
    SMode7Sel := false;
    SAnyModeSel := false;
    Error := false;
16#8005:
    Ready := true;
    SMode0Sel := false;
    SMode1Sel := false;
    SMode2Sel := false;
    SMode3Sel := false;
    SMode4Sel := false;
    SMode5Sel := false;
    SMode6Sel := false;
    SMode7Sel := false;
    SAnyModeSel := false;
    Error := false;
16#8000:
    Ready := true;
    SMode0Sel := SMode0;
    SMode1Sel := SMode1;
    SMode2Sel := SMode2;
    SMode3Sel := SMode3;
    SMode4Sel := SMode4;
    SMode5Sel := SMode5;
    SMode6Sel := SMode6;
    SMode7Sel := SMode7;
    SAnyModeSel := true;
    Error := false;
16#8004:
    Ready := true;
    SAnyModeSel := true;
    Error := false;
16#C001,
16#C002,
16#C003,
16#C004:
    Ready := true;
    SMode0Sel := false;
    SMode1Sel := false;
    SMode2Sel := false;
    SMode3Sel := false;
    SMode4Sel := false;
    SMode5Sel := false;
    SMode6Sel := false;
    SMode7Sel := false;
    SAnyModeSel := false;
    Error := true;
END_CASE;
IF (DiagCode <> 16#8005) THEN
    IN:=FALSE;
    PT:=ModeMonitorTime;
    Q := FALSE;
    running := FALSE;
END_IF;
END_FUNCTION_BLOCK

(* ---- SFModeSelector_CAP.st ---- *)
PROGRAM Main
VAR_INPUT
    Activate : BOOL;
    SMode0 : BOOL;
    SMode1 : BOOL;
    SMode2 : BOOL;
    SMode3 : BOOL;
    SMode4 : BOOL;
    SMode5 : BOOL;
    SMode6 : BOOL;
    SMode7 : BOOL;
    SUnlock : BOOL;
    SSetMode : BOOL;
    AutoSetMode : BOOL;
    ModeMonitorTime : TIME;
    Reset : BOOL;
END_VAR
VAR
    SFModeSelector : SFModeSelector;
END_VAR
SFModeSelector(Activate:=Activate,SMode0:=SMode0,SMode1:=SMode1,SMode2:=SMode2,SMode3:=SMode3,SMode4:=SMode4,SMode5:=SMode5,
SMode6:=SMode6,SMode7:=SMode7,SUnlock:=SUnlock,SSetMode:=SSetMode,AutoSetMode:=AutoSetMode,ModeMonitorTime:=ModeMonitorTime,
Reset:=Reset);
END_PROGRAM

FUNCTION_BLOCK SFModeSelector
VAR_INPUT
    Activate : BOOL;
    SMode0 : BOOL;
    SMode1 : BOOL;
    SMode2 : BOOL;
    SMode3 : BOOL;
    SMode4 : BOOL;
    SMode5 : BOOL;
    SMode6 : BOOL;
    SMode7 : BOOL;
    SUnlock : BOOL;
    SSetMode : BOOL;
    AutoSetMode : BOOL;
    ModeMonitorTime : TIME;
    Reset : BOOL;
END_VAR
VAR
    IN : BOOL;
    PT : TIME;
    running : BOOL;
    Q : BOOL;
    RTRIGatResetQ : BOOL;
    RTRIGatResetM : BOOL;
    RTRIGatSetModeQ : BOOL;
    RTRIGatSetModeM : BOOL;
    FTRIGatModeSel0Q : BOOL;
    FTRIGatModeSel0M : BOOL;
    RTRIGatModeSel0Q: BOOL;
    RTRIGatModeSel0M: BOOL;
    fallingEdgeDetected : BOOL;
END_VAR
VAR_TEMP
    Error1 : BOOL;
    Error2 : BOOL;
END_VAR
VAR_OUTPUT
    Ready : BOOL;
    SMode0Sel : BOOL;
    SMode1Sel : BOOL;
    SMode2Sel : BOOL;
    SMode3Sel : BOOL;
    SMode4Sel : BOOL;
    SMode5Sel : BOOL;
    SMode6Sel : BOOL;
    SMode7Sel : BOOL;
    SAnyModeSel : BOOL;
    Error : BOOL;
    DiagCode : WORD;
END_VAR
RTRIGatResetQ := Reset AND NOT RTRIGatResetM;
RTRIGatResetM := Reset;

RTRIGatSetModeQ := SSetMode AND NOT RTRIGatSetModeM;
RTRIGatSetModeM := SSetMode;

IF NOT Activate THEN
    DiagCode := 16#0000;
ELSE
    IF (SMode0 + SMode1 + SMode2 + SMode3 + SMode4 + SMode5 + SMode6 + SMode7 > 1) THEN
        Error1 := true;
    ELSE
        Error1 := false;
    END_IF;
    CASE DiagCode OF
    16#0000:
        IF Activate THEN
            DiagCode := 16#8005;
        END_IF;
    16#8005:
        IF (NOT SMode0 AND NOT SMode1 AND NOT SMode2 AND NOT SMode3 AND NOT SMode4 AND NOT SMode5 AND NOT SMode6 AND NOT SMode7) THEN
            FTRIGatModeSel0Q := NOT false AND FTRIGatModeSel0M;
            FTRIGatModeSel0M := false;
            RTRIGatModeSel0Q := false AND NOT RTRIGatModeSel0M;
            RTRIGatModeSel0M := false;
        ELSE
            FTRIGatModeSel0Q := NOT true AND FTRIGatModeSel0M;
            FTRIGatModeSel0M := true;
            RTRIGatModeSel0Q := true AND NOT RTRIGatModeSel0M;
            RTRIGatModeSel0M := true;
        END_IF;
        IF FTRIGatModeSel0Q THEN
            fallingEdgeDetected := TRUE;
        END_IF;
        IF fallingEdgeDetected THEN
            IN:=TRUE;
            PT:=ModeMonitorTime;
            IF NOT running AND NOT Q THEN
                running := TRUE;
            ELSIF running AND NOT Q THEN
                Q := NONDETERMINISTIC_BOOL();
                running := NOT Q;
            END_IF;
        ELSIF RTRIGatModeSel0Q THEN
            IN:=FALSE;
            PT:=ModeMonitorTime;
            Q := FALSE;
            running := FALSE;
            fallingEdgeDetected := FALSE;
        END_IF;
        Error2 := Q;
        IF Error1 THEN
            DiagCode := 16#C001;
        ELSIF Error2 THEN
            DiagCode := 16#C002;
        ELSIF ((AutoSetMode OR RTRIGatSetModeQ) AND SUnlock AND (SMode0 + SMode1 + SMode2 + SMode3 + SMode4 + SMode5 + SMode6 + SMode7 = 1)) THEN
            DiagCode := 16#8000;
        END_IF;
    16#8000:
        IF Error1 THEN
            DiagCode := 16#C001;
        ELSIF (SMode0 <> SMode0Sel OR SMode1 <> SMode1Sel OR SMode2 <> SMode2Sel OR SMode3 <> SMode3Sel
              OR SMode4 <> SMode4Sel OR SMode5 <> SMode5Sel OR SMode6 <> SMode6Sel OR SMode7 <> SMode7Sel) THEN
            DiagCode := 16#8005;
            fallingEdgeDetected := FALSE;
        ELSIF (NOT SUnlock) THEN
            DiagCode := change(16#8004, 16#8000);
        END_IF;
    16#8004:
        IF SUnlock THEN
            DiagCode := 16#8000;
        END_IF;
    16#C001:
        IF Reset AND NOT RTRIGatResetQ THEN
            DiagCode := 16#C003;
        ELSIF RTRIGatResetQ THEN
            DiagCode := 16#8005;
            fallingEdgeDetected := FALSE;
        END_IF;
    16#C002:
        IF Reset AND NOT RTRIGatResetQ THEN
            DiagCode := 16#C004;
        ELSIF RTRIGatResetQ THEN
            DiagCode := 16#8005;
            fallingEdgeDetected := FALSE;
        END_IF;
    16#C003:
        IF (NOT Reset) THEN
            DiagCode := 16#C001;
        END_IF;
    16#C004:
        IF (NOT Reset) THEN
            DiagCode := 16#C002;
        END_IF;
    END_CASE;
END_IF;

CASE DiagCode OF
16#0000:
    Ready := false;
    SMode0Sel := false;
    SMode1Sel := false;
    SMode2Sel := false;
    SMode3Sel := false;
    SMode4Sel := false;
    SMode5Sel := false;
    SMode6Sel := false;
    SMode7Sel := false;
    SAnyModeSel := false;
    Error := false;
16#8005:
    Ready := true;
    SMode0Sel := false;
    SMode1Sel := false;
    SMode2Sel := false;
    SMode3Sel := false;
    SMode4Sel := false;
    SMode5Sel := false;
    SMode6Sel := false;
    SMode7Sel := false;
    SAnyModeSel := false;
    Error := false;
16#8000:
    Ready := true;
    SMode0Sel := SMode0;
    SMode1Sel := SMode1;
    SMode2Sel := SMode2;
    SMode3Sel := SMode3;
    SMode4Sel := SMode4;
    SMode5Sel := SMode5;
    SMode6Sel := SMode6;
    SMode7Sel := SMode7;
    SAnyModeSel := true;
    Error := false;
16#8004:
    Ready := true;
    SAnyModeSel := true;
    Error := false;
16#C001,
16#C002,
16#C003,
16#C004:
    Ready := true;
    SMode0Sel := false;
    SMode1Sel := false;
    SMode2Sel := false;
    SMode3Sel := false;
    SMode4Sel := false;
    SMode5Sel := false;
    SMode6Sel := false;
    SMode7Sel := false;
    SAnyModeSel := false;
    Error := true;
END_CASE;
IF (DiagCode <> 16#8005) THEN
    IN:=FALSE;
    PT:=ModeMonitorTime;
    Q := FALSE;
    running := FALSE;
END_IF;
END_FUNCTION_BLOCK

(* ---- SFMutingSeq.st ---- *)
PROGRAM Main
VAR_INPUT
    Activate : BOOL := FALSE;
    SAOPDIn : SAFEBOOL := FALSE;
    MutingSwitch11 : BOOL := FALSE;
    MutingSwitch12 : BOOL := FALSE;
    MutingSwitch21 : BOOL := FALSE;
    MutingSwitch22 : BOOL := FALSE;
    SMutingLamp : SAFEBOOL := FALSE;
    DiscTime1112 : TIME := T#0s;
    DiscTime2122 : TIME := T#0s;
    MaxMutingTime : TIME := T#0s;
    MutingEnable : BOOL := FALSE;
    SStartReset : SAFEBOOL := FALSE;
    Reset : BOOL := FALSE;
END_VAR
VAR
    SFMutingSeq : SFMutingSeq;
END_VAR
SFMutingSeq(Activate:=Activate,SAOPDIn:=SAOPDIn,MutingSwitch11:=MutingSwitch11,MutingSwitch12:=MutingSwitch12,MutingSwitch21:=MutingSwitch21,
MutingSwitch22:=MutingSwitch22,SMutingLamp:=SMutingLamp,DiscTime1112:=DiscTime1112,DiscTime2122:=DiscTime2122,
MaxMutingTime:=MaxMutingTime,MutingEnable:=MutingEnable,SStartReset:=SStartReset,Reset:=Reset);
END_PROGRAM

FUNCTION_BLOCK SFMutingSeq
VAR_INPUT
    Activate : BOOL := FALSE;
    SAOPDIn : SAFEBOOL := FALSE;
    MutingSwitch11 : BOOL := FALSE;
    MutingSwitch12 : BOOL := FALSE;
    MutingSwitch21 : BOOL := FALSE;
    MutingSwitch22 : BOOL := FALSE;
    SMutingLamp : SAFEBOOL := FALSE;
    DiscTime1112 : TIME := T#0s;
    DiscTime2122 : TIME := T#0s;
    MaxMutingTime : TIME := T#0s;
    MutingEnable : BOOL := FALSE;
    SStartReset : SAFEBOOL := FALSE;
    Reset : BOOL := FALSE;
END_VAR
VAR
    IN : BOOL;
    PT : TIME;
    running : BOOL;
    Q : BOOL;
    RTRIGatResetQ : BOOL;
    RTRIGatResetM : BOOL;
    RTRIGatMS11Q : BOOL;
    RTRIGatMS11M : BOOL;
    RTRIGatMS12Q : BOOL;
    RTRIGatMS12M : BOOL;
    RTRIGatMS21Q : BOOL;
    RTRIGatMS21M : BOOL;
    RTRIGatMS22Q : BOOL;
    RTRIGatMS22M : BOOL;
    FTRIGatMS11Q : BOOL;
    FTRIGatMS11M : BOOL;
    FTRIGatMS12Q : BOOL;
    FTRIGatMS12M : BOOL;
    FTRIGatMS21Q : BOOL;
    FTRIGatMS21M : BOOL;
    FTRIGatMS22Q : BOOL;
    FTRIGatMS22M : BOOL;
END_VAR
VAR_OUTPUT
    Ready : BOOL := FALSE;
    SAOPDOut : SAFEBOOL := FALSE;
    SMutingActive : SAFEBOOL := FALSE;
    Error : BOOL := FALSE;
    DiagCode : WORD := 16#0000;
END_VAR
RTRIGatResetQ := Reset AND NOT RTRIGatResetM;
RTRIGatResetM := Reset;

RTRIGatMS11Q := MutingSwitch11 AND NOT RTRIGatMS11M;
RTRIGatMS11M := MutingSwitch11;

RTRIGatMS12Q := MutingSwitch12 AND NOT RTRIGatMS12M;
RTRIGatMS12M := MutingSwitch12;

RTRIGatMS21Q := MutingSwitch21 AND NOT RTRIGatMS21M;
RTRIGatMS21M := MutingSwitch21;

RTRIGatMS22Q := MutingSwitch22 AND NOT RTRIGatMS22M;
RTRIGatMS22M := MutingSwitch22;

FTRIGatMS11Q := NOT MutingSwitch11 AND FTRIGatMS11M;
FTRIGatMS11M := MutingSwitch11;

FTRIGatMS12Q := NOT MutingSwitch12 AND FTRIGatMS12M;
FTRIGatMS12M := MutingSwitch12;

FTRIGatMS21Q := NOT MutingSwitch21 AND FTRIGatMS21M;
FTRIGatMS21M := MutingSwitch21;

FTRIGatMS22Q := NOT MutingSwitch22 AND FTRIGatMS22M;
FTRIGatMS22M := MutingSwitch22;

IF NOT Activate THEN
    DiagCode := 16#0000;
ELSE
    CASE DiagCode OF
    16#0000:
    IF Activate THEN
        DiagCode := 16#8001;
    END_IF;
    16#8000:
        IF (NOT MutingEnable AND RTRIGatMS11Q) OR (NOT MutingEnable AND RTRIGatMS22Q) OR (MutingSwitch12 OR MutingSwitch21) OR (MutingSwitch11 AND MutingSwitch22) THEN
            (* Wrong muting sequence *)
            DiagCode := 16#C004;
        ELSIF NOT SAOPDIn THEN
            DiagCode := 16#8002;
        ELSIF NOT SMutingLamp THEN
            DiagCode := 16#C003;
        ELSIF MutingEnable AND (RTRIGatMS11Q AND NOT MutingSwitch12 AND NOT MutingSwitch21 AND NOT MutingSwitch22) THEN
            DiagCode := 16#8011;
            IN:=TRUE;
            PT:=MaxMutingTime;
            IF NOT running AND NOT Q THEN
                running := TRUE;
            ELSIF running AND NOT Q THEN
                Q := NONDETERMINISTIC_BOOL();
                running := NOT Q;
            END_IF;
        ELSIF MutingEnable AND (NOT MutingSwitch11 AND NOT MutingSwitch12 AND NOT MutingSwitch21 AND RTRIGatMS22Q) THEN
            DiagCode := 16#8122;
            IN:=TRUE;
            PT:=MaxMutingTime;
            IF NOT running AND NOT Q THEN
                running := TRUE;
            ELSIF running AND NOT Q THEN
                Q := NONDETERMINISTIC_BOOL();
                running := NOT Q;
            END_IF;
        END_IF;
    16#8001:
        IF Reset AND NOT RTRIGatResetQ AND NOT SStartReset THEN
            DiagCode := 16#C001;
        (*
        ELSIF (Time parameters out of range)
        DiagCode := 16#C005;
        *)
        ELSIF RTRIGatResetQ OR SStartReset THEN
            DiagCode := 16#8005;
        END_IF;
    16#8002:
        IF SAOPDIn THEN
            DiagCode := 16#8003;
        END_IF;
    16#8003:
        IF Reset AND NOT RTRIGatResetQ THEN
            DiagCode := 16#C002;
        ELSIF RTRIGatResetQ THEN
            DiagCode := 16#8005;
        END_IF;
    16#8005:
        IF NOT SAOPDIn THEN
            DiagCode := 16#8002;
        ELSIF NOT SMutingLamp THEN
            DiagCode := 16#C003;
        ELSIF SAOPDIn THEN
            DiagCode := 16#8000;
        END_IF;
    16#C001:
        IF NOT Reset THEN
            DiagCode := 16#8001;
        END_IF;
    16#C002:
        IF NOT Reset THEN
            DiagCode := 16#8003;
        END_IF;
    16#C003:
        IF SMutingLamp THEN
            DiagCode := 16#8003;
        END_IF;
    16#C006,
    16#C007,
    16#C008:
        IF NOT (MutingSwitch11 OR MutingSwitch12 OR MutingSwitch21 OR MutingSwitch22) THEN
            DiagCode := 16#8003;
        END_IF;
    ELSE
        IF DiagCode >= 16#C000 THEN
        (* 16#CYx4 *)
            IF NOT (MutingSwitch11 OR MutingSwitch12 OR MutingSwitch21 OR MutingSwitch22) THEN
                DiagCode := 16#8003;
            END_IF;
        ELSE
            (* cases 16#8011 .. 16#8422 *)
            CASE DiagCode OF
            16#8011:
                IF NOT MutingEnable OR NOT MutingSwitch11 OR MutingSwitch21 OR MutingSwitch22 THEN
                    DiagCode := 16#C104;
                ELSIF Q THEN
                    DiagCode := 16#C006;
                ELSIF NOT SAOPDIn THEN
                    DiagCode := 16#8002;
                ELSIF NOT SMutingLamp THEN
                    DiagCode := 16#C003;
                ELSIF MutingEnable AND (MutingSwitch11 AND RTRIGatMS12Q AND NOT MutingSwitch21 AND NOT MutingSwitch22) THEN
                    DiagCode := 16#8012;
                END_IF;
            16#8012:
                IF RTRIGatMS11Q OR RTRIGatMS12Q OR FTRIGatMS22Q THEN
                    DiagCode := 16#C104;
                ELSIF Q THEN
                    DiagCode := 16#C006;
                ELSIF NOT SMutingLamp THEN
                    DiagCode := 16#C003;
                ELSIF NOT MutingSwitch11 AND NOT MutingSwitch12 AND FTRIGatMS21Q AND MutingSwitch22 THEN
                    IN:=FALSE;
                    PT:=MaxMutingTime;
                    Q := FALSE;
                    running := FALSE;
                    DiagCode := 16#8000;
                END_IF;
            16#8122:
                IF NOT MutingEnable OR MutingSwitch11 OR MutingSwitch12 OR NOT MutingSwitch22 THEN
                    DiagCode := 16#C104;
                ELSIF Q THEN
                    DiagCode := 16#C006;
                ELSIF NOT SAOPDIn THEN
                    DiagCode := 16#8002;
                ELSIF NOT SMutingLamp THEN
                    DiagCode := 16#C003;
                ELSIF MutingEnable AND (NOT MutingSwitch11 AND NOT MutingSwitch12 AND RTRIGatMS21Q AND MutingSwitch22) THEN
                    DiagCode := 16#8112;
                END_IF;
            16#8112:
                IF FTRIGatMS11Q OR RTRIGatMS21Q OR RTRIGatMS22Q THEN
                    DiagCode := 16#C104;
                ELSIF Q THEN
                    DiagCode := 16#C006;
                ELSIF NOT SMutingLamp THEN
                    DiagCode := 16#C003;
                ELSIF MutingSwitch11 AND FTRIGatMS12Q AND NOT MutingSwitch21 AND NOT MutingSwitch22 THEN
                    DiagCode := 16#8000;
                    IN:=FALSE;
                    PT:=MaxMutingTime;
                    Q := FALSE;
                    running := FALSE;
                END_IF;
            END_CASE;
        END_IF;
    END_CASE;
END_IF;
CASE DiagCode OF
16#0000:
    Ready := FALSE;
    SAOPDOut := FALSE;
    SMutingActive := FALSE;
    Error := FALSE;
16#8000,
16#8011,
16#8122:
    Ready := TRUE;
    SAOPDOut := TRUE;
    SMutingActive := FALSE;
    Error := FALSE;
16#8001,
16#8002,
16#8003,
16#8005:
    Ready := TRUE;
    SAOPDOut := FALSE;
    SMutingActive := FALSE;
    Error := FALSE;
16#8012,
16#8112:
    Ready := TRUE;
    SAOPDOut := TRUE;
    SMutingActive := TRUE;
    Error := FALSE;
ELSE
    Ready := TRUE;
    SAOPDOut := FALSE;
    SMutingActive := FALSE;
    Error := TRUE;
END_CASE;
END_FUNCTION_BLOCK

(* ---- SFMutingSeq_CAP.st ---- *)
PROGRAM Main
VAR_INPUT
    Activate : BOOL := FALSE;
    SAOPDIn : SAFEBOOL := FALSE;
    MutingSwitch11 : BOOL := FALSE;
    MutingSwitch12 : BOOL := FALSE;
    MutingSwitch21 : BOOL := FALSE;
    MutingSwitch22 : BOOL := FALSE;
    SMutingLamp : SAFEBOOL := FALSE;
    DiscTime1112 : TIME := T#0s;
    DiscTime2122 : TIME := T#0s;
    MaxMutingTime : TIME := T#0s;
    MutingEnable : BOOL := FALSE;
    SStartReset : SAFEBOOL := FALSE;
    Reset : BOOL := FALSE;
END_VAR
VAR
    SFMutingSeq : SFMutingSeq;
END_VAR
SFMutingSeq(Activate:=Activate,SAOPDIn:=SAOPDIn,MutingSwitch11:=MutingSwitch11,MutingSwitch12:=MutingSwitch12,MutingSwitch21:=MutingSwitch21,
MutingSwitch22:=MutingSwitch22,SMutingLamp:=SMutingLamp,DiscTime1112:=DiscTime1112,DiscTime2122:=DiscTime2122,
MaxMutingTime:=MaxMutingTime,MutingEnable:=MutingEnable,SStartReset:=SStartReset,Reset:=Reset);
END_PROGRAM

FUNCTION_BLOCK SFMutingSeq
VAR_INPUT
    Activate : BOOL := FALSE;
    SAOPDIn : SAFEBOOL := FALSE;
    MutingSwitch11 : BOOL := FALSE;
    MutingSwitch12 : BOOL := FALSE;
    MutingSwitch21 : BOOL := FALSE;
    MutingSwitch22 : BOOL := FALSE;
    SMutingLamp : SAFEBOOL := FALSE;
    DiscTime1112 : TIME := T#0s;
    DiscTime2122 : TIME := T#0s;
    MaxMutingTime : TIME := T#0s;
    MutingEnable : BOOL := FALSE;
    SStartReset : SAFEBOOL := FALSE;
    Reset : BOOL := FALSE;
END_VAR
VAR
    IN : BOOL;
    PT : TIME;
    running : BOOL;
    Q : BOOL;
    RTRIGatResetQ : BOOL;
    RTRIGatResetM : BOOL;
    RTRIGatMS11Q : BOOL;
    RTRIGatMS11M : BOOL;
    RTRIGatMS12Q : BOOL;
    RTRIGatMS12M : BOOL;
    RTRIGatMS21Q : BOOL;
    RTRIGatMS21M : BOOL;
    RTRIGatMS22Q : BOOL;
    RTRIGatMS22M : BOOL;
    FTRIGatMS11Q : BOOL;
    FTRIGatMS11M : BOOL;
    FTRIGatMS12Q : BOOL;
    FTRIGatMS12M : BOOL;
    FTRIGatMS21Q : BOOL;
    FTRIGatMS21M : BOOL;
    FTRIGatMS22Q : BOOL;
    FTRIGatMS22M : BOOL;
END_VAR
VAR_OUTPUT
    Ready : BOOL := FALSE;
    SAOPDOut : SAFEBOOL := FALSE;
    SMutingActive : SAFEBOOL := FALSE;
    Error : BOOL := FALSE;
    DiagCode : WORD := 16#0000;
END_VAR
RTRIGatResetQ := Reset AND NOT RTRIGatResetM;
RTRIGatResetM := Reset;

RTRIGatMS11Q := MutingSwitch11 AND NOT RTRIGatMS11M;
RTRIGatMS11M := MutingSwitch11;

RTRIGatMS12Q := MutingSwitch12 AND NOT RTRIGatMS12M;
RTRIGatMS12M := MutingSwitch12;

RTRIGatMS21Q := MutingSwitch21 AND NOT RTRIGatMS21M;
RTRIGatMS21M := MutingSwitch21;

RTRIGatMS22Q := MutingSwitch22 AND NOT RTRIGatMS22M;
RTRIGatMS22M := MutingSwitch22;

FTRIGatMS11Q := NOT MutingSwitch11 AND FTRIGatMS11M;
FTRIGatMS11M := MutingSwitch11;

FTRIGatMS12Q := NOT MutingSwitch12 AND FTRIGatMS12M;
FTRIGatMS12M := MutingSwitch12;

FTRIGatMS21Q := NOT MutingSwitch21 AND FTRIGatMS21M;
FTRIGatMS21M := MutingSwitch21;

FTRIGatMS22Q := NOT MutingSwitch22 AND FTRIGatMS22M;
FTRIGatMS22M := MutingSwitch22;

IF NOT Activate THEN
    DiagCode := 16#0000;
ELSE
    CASE DiagCode OF
    16#0000:
    IF Activate THEN
        DiagCode := 16#8001;
    END_IF;
    16#8000:
        IF (NOT MutingEnable AND RTRIGatMS11Q) OR (NOT MutingEnable AND RTRIGatMS22Q) OR (MutingSwitch12 OR MutingSwitch21) OR (MutingSwitch11 AND MutingSwitch22) THEN
            (* Wrong muting sequence *)
            DiagCode := 16#C004;
        ELSIF NOT SAOPDIn THEN
            DiagCode := 16#8002;
        ELSIF NOT SMutingLamp THEN
            DiagCode := 16#C003;
        ELSIF MutingEnable AND (RTRIGatMS11Q AND NOT MutingSwitch12 AND NOT MutingSwitch21 AND NOT MutingSwitch22) THEN
            DiagCode := change(16#8011, 16#8005);
            IN:=TRUE;
            PT:=MaxMutingTime;
            IF NOT running AND NOT Q THEN
                running := TRUE;
            ELSIF running AND NOT Q THEN
                Q := NONDETERMINISTIC_BOOL();
                running := NOT Q;
            END_IF;
        ELSIF MutingEnable AND (NOT MutingSwitch11 AND NOT MutingSwitch12 AND NOT MutingSwitch21 AND RTRIGatMS22Q) THEN
            DiagCode := 16#8122;
            IN:=TRUE;
            PT:=MaxMutingTime;
            IF NOT running AND NOT Q THEN
                running := TRUE;
            ELSIF running AND NOT Q THEN
                Q := NONDETERMINISTIC_BOOL();
                running := NOT Q;
            END_IF;
        END_IF;
    16#8001:
        IF Reset AND NOT RTRIGatResetQ AND NOT SStartReset THEN
            DiagCode := 16#C001;
        (*
        ELSIF (Time parameters out of range)
        DiagCode := 16#C005;
        *)
        ELSIF RTRIGatResetQ OR SStartReset THEN
            DiagCode := 16#8005;
        END_IF;
    16#8002:
        IF SAOPDIn THEN
            DiagCode := 16#8003;
        END_IF;
    16#8003:
        IF Reset AND NOT RTRIGatResetQ THEN
            DiagCode := 16#C002;
        ELSIF RTRIGatResetQ THEN
            DiagCode := 16#8005;
        END_IF;
    16#8005:
        IF NOT SAOPDIn THEN
            DiagCode := 16#8002;
        ELSIF NOT SMutingLamp THEN
            DiagCode := 16#C003;
        ELSIF SAOPDIn THEN
            DiagCode := 16#8000;
        END_IF;
    16#C001:
        IF NOT Reset THEN
            DiagCode := 16#8001;
        END_IF;
    16#C002:
        IF NOT Reset THEN
            DiagCode := 16#8003;
        END_IF;
    16#C003:
        IF SMutingLamp THEN
            DiagCode := 16#8003;
        END_IF;
    16#C006,
    16#C007,
    16#C008:
        IF NOT (MutingSwitch11 OR MutingSwitch12 OR MutingSwitch21 OR MutingSwitch22) THEN
            DiagCode := 16#8003;
        END_IF;
    ELSE
        IF DiagCode >= 16#C000 THEN
        (* 16#CYx4 *)
            IF NOT (MutingSwitch11 OR MutingSwitch12 OR MutingSwitch21 OR MutingSwitch22) THEN
                DiagCode := 16#8003;
            END_IF;
        ELSE
            (* cases 16#8011 .. 16#8422 *)
            CASE DiagCode OF
            16#8011:
                IF NOT MutingEnable OR NOT MutingSwitch11 OR MutingSwitch21 OR MutingSwitch22 THEN
                    DiagCode := 16#C104;
                ELSIF Q THEN
                    DiagCode := 16#C006;
                ELSIF NOT SAOPDIn THEN
                    DiagCode := 16#8002;
                ELSIF NOT SMutingLamp THEN
                    DiagCode := 16#C003;
                ELSIF MutingEnable AND (MutingSwitch11 AND RTRIGatMS12Q AND NOT MutingSwitch21 AND NOT MutingSwitch22) THEN
                    DiagCode := 16#8012;
                END_IF;
            16#8012:
                IF RTRIGatMS11Q OR RTRIGatMS12Q OR FTRIGatMS22Q THEN
                    DiagCode := 16#C104;
                ELSIF Q THEN
                    DiagCode := 16#C006;
                ELSIF NOT SMutingLamp THEN
                    DiagCode := 16#C003;
                ELSIF NOT MutingSwitch11 AND NOT MutingSwitch12 AND FTRIGatMS21Q AND MutingSwitch22 THEN
                    IN:=FALSE;
                    PT:=MaxMutingTime;
                    Q := FALSE;
                    running := FALSE;
                    DiagCode := 16#8000;
                END_IF;
            16#8122:
                IF NOT MutingEnable OR MutingSwitch11 OR MutingSwitch12 OR NOT MutingSwitch22 THEN
                    DiagCode := 16#C104;
                ELSIF Q THEN
                    DiagCode := 16#C006;
                ELSIF NOT SAOPDIn THEN
                    DiagCode := 16#8002;
                ELSIF NOT SMutingLamp THEN
                    DiagCode := 16#C003;
                ELSIF MutingEnable AND (NOT MutingSwitch11 AND NOT MutingSwitch12 AND RTRIGatMS21Q AND MutingSwitch22) THEN
                    DiagCode := 16#8112;
                END_IF;
            16#8112:
                IF FTRIGatMS11Q OR RTRIGatMS21Q OR RTRIGatMS22Q THEN
                    DiagCode := 16#C104;
                ELSIF Q THEN
                    DiagCode := 16#C006;
                ELSIF NOT SMutingLamp THEN
                    DiagCode := 16#C003;
                ELSIF MutingSwitch11 AND FTRIGatMS12Q AND NOT MutingSwitch21 AND NOT MutingSwitch22 THEN
                    DiagCode := 16#8000;
                    IN:=FALSE;
                    PT:=MaxMutingTime;
                    Q := FALSE;
                    running := FALSE;
                END_IF;
            END_CASE;
        END_IF;
    END_CASE;
END_IF;
CASE DiagCode OF
16#0000:
    Ready := FALSE;
    SAOPDOut := FALSE;
    SMutingActive := FALSE;
    Error := FALSE;
16#8000,
16#8011,
16#8122:
    Ready := TRUE;
    SAOPDOut := TRUE;
    SMutingActive := FALSE;
    Error := FALSE;
16#8001,
16#8002,
16#8003,
16#8005:
    Ready := TRUE;
    SAOPDOut := FALSE;
    SMutingActive := FALSE;
    Error := FALSE;
16#8012,
16#8112:
    Ready := TRUE;
    SAOPDOut := TRUE;
    SMutingActive := TRUE;
    Error := FALSE;
ELSE
    Ready := TRUE;
    SAOPDOut := FALSE;
    SMutingActive := FALSE;
    Error := TRUE;
END_CASE;
END_FUNCTION_BLOCK
